KUKA KRL program: MyProgram_152().src

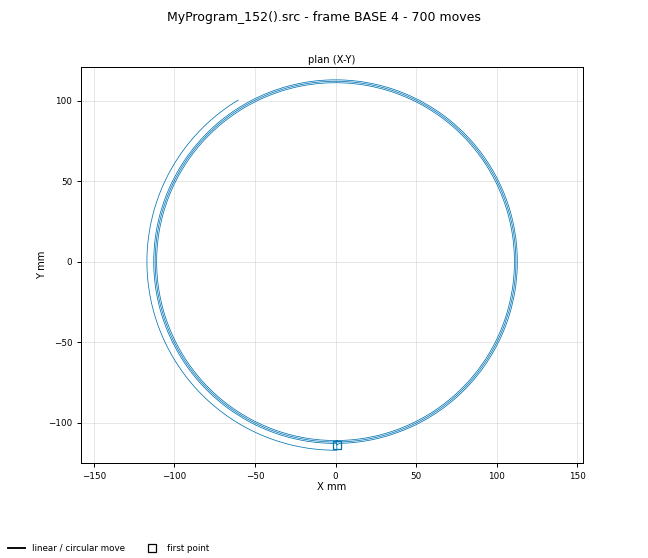
[picture p0: tool path of MyProgram_152().src in frame BASE 4, 700 of 700 moves have a stored position in this frame; points joined in program order, loops and branches not executed]
&ACCESS RVP
&REL 1
&PARAM TEMPLATE = C:\KRC\Roboter\Template\vorgabe
&PARAM EDITMASK = *
DEF MyProgram_152()
; ---- Setting reference (Base) ----
$BASE = BASE_DATA[4]

; --------------------------
; ---- Setting tool (TCP) ----
$TOOL = TOOL_DATA[3]
; --------------------------

$VEL.CP = VEL_APROX_PRINT
LIN {X 0.8048,Y -113.7717,Z 118,A -93.5748,B 24.9556,C -1.539,E1 25.0005,E2 539.5686} C_DIS
Startdeposition()
$VEL.CP = VEL_PRINT
LIN {X 2.402,Y -112.8589,Z 118,A -92.1297,B 24.9531,C -1.5823,E1 25.0048,E2 538.0211} C_DIS
LIN {X 9.2872,Y -112.5017,Z 118,A -88.8373,B 24.9535,C -1.5747,E1 25.014,E2 534.748} C_DIS
LIN {X 15.0576,Y -111.8766,Z 118,A -85.7735,B 24.9531,C -1.5815,E1 25.0225,E2 531.6701} C_DIS
LIN {X 17.7675,Y -111.4782,Z 118,A -84.0166,B 24.9521,C -1.5987,E1 25.0275,E2 529.8742} C_DIS
LIN {X 21.9684,Y -110.727,Z 118,A -81.6298,B 24.9514,C -1.6103,E1 25.0341,E2 527.4627} C_DIS
LIN {X 25.6031,Y -109.9423,Z 118,A -80.4099,B 24.9531,C -1.5825,E1 25.0372,E2 526.3104} C_DIS
LIN {X 28.0521,Y -109.3429,Z 118,A -78.9806,B 24.9526,C -1.5904,E1 25.0411,E2 524.8645} C_DIS
LIN {X 31.4481,Y -108.4172,Z 118,A -77.0293,B 24.9521,C -1.5997,E1 25.0464,E2 522.8944} C_DIS
LIN {X 34.8547,Y -107.3683,Z 118,A -75.3553,B 24.9523,C -1.5959,E1 25.0508,E2 521.2326} C_DIS
LIN {X 42.209,Y -104.6964,Z 118,A -70.4589,B 24.9494,C -1.643,E1 25.0639,E2 516.2353} C_DIS
LIN {X 47.5182,Y -102.3955,Z 118,A -68.4504,B 24.9517,C -1.6055,E1 25.0687,E2 514.3206} C_DIS
LIN {X 50.4487,Y -100.9844,Z 118,A -66.7644,B 24.9514,C -1.6098,E1 25.073,E2 512.6289} C_DIS
LIN {X 54.4638,Y -98.8775,Z 118,A -64.3708,B 24.9509,C -1.6179,E1 25.0789,E2 510.2228} C_DIS
LIN {X 57.7854,Y -96.9732,Z 118,A -62.5355,B 24.951,C -1.6166,E1 25.0833,E2 508.3961} C_DIS
LIN {X 62.6769,Y -93.8871,Z 118,A -59.5043,B 24.9504,C -1.6267,E1 25.0904,E2 505.3512} C_DIS
LIN {X 66.3277,Y -91.3435,Z 118,A -57.343,B 24.9504,C -1.627,E1 25.0953,E2 503.1967} C_DIS
LIN {X 69.139,Y -89.2339,Z 118,A -55.545,B 24.9501,C -1.6315,E1 25.0993,E2 501.3946} C_DIS
LIN {X 72.1712,Y -86.7993,Z 118,A -53.7011,B 24.9502,C -1.63,E1 25.1033,E2 499.5613} C_DIS
LIN {X 75.0077,Y -84.361,Z 118,A -51.7648,B 24.9498,C -1.6361,E1 25.1074,E2 497.6182} C_DIS
LIN {X 77.4909,Y -82.0853,Z 118,A -50.0402,B 24.9495,C -1.6409,E1 25.1109,E2 495.8893} C_DIS
LIN {X 80.3457,Y -79.2929,Z 118,A -48.1006,B 24.9495,C -1.6418,E1 25.1147,E2 493.9557} C_DIS
LIN {X 82.9222,Y -76.5954,Z 118,A -46.1586,B 24.9491,C -1.6488,E1 25.1185,E2 492.0056} C_DIS
LIN {X 85.1759,Y -74.0805,Z 118,A -44.45,B 24.9488,C -1.653,E1 25.1216,E2 490.2948} C_DIS
LIN {X 87.7234,Y -71.045,Z 118,A -42.5175,B 24.9487,C -1.6548,E1 25.125,E2 488.3671} C_DIS
LIN {X 89.93,Y -68.2326,Z 118,A -40.2028,B 24.9469,C -1.6828,E1 25.1291,E2 485.9971} C_DIS
LIN {X 92.1441,Y -65.2094,Z 118,A -38.7629,B 24.9479,C -1.6667,E1 25.1313,E2 484.6022} C_DIS
LIN {X 93.913,Y -62.6378,Z 118,A -36.957,B 24.947,C -1.6814,E1 25.1342,E2 482.7706} C_DIS
LIN {X 97.4321,Y -57.009,Z 118,A -33.6398,B 24.9466,C -1.6888,E1 25.139,E2 479.453} C_DIS
LIN {X 99.7325,Y -52.8802,Z 118,A -31.4879,B 24.9468,C -1.6844,E1 25.1418,E2 477.3226} C_DIS
LIN {X 101.2277,Y -49.9579,Z 118,A -29.5164,B 24.9456,C -1.7037,E1 25.1443,E2 475.3163} C_DIS
LIN {X 102.6063,Y -47.0654,Z 118,A -28.3237,B 24.9466,C -1.6884,E1 25.1457,E2 474.166} C_DIS
LIN {X 104.8738,Y -41.7679,Z 118,A -25.458,B 24.9462,C -1.6947,E1 25.1488,E2 471.3012} C_DIS
LIN {X 106.2374,Y -38.167,Z 118,A -23.2124,B 24.9449,C -1.7143,E1 25.151,E2 469.0218} C_DIS
LIN {X 107.3896,Y -34.7888,Z 118,A -21.1915,B 24.9439,C -1.7299,E1 25.1528,E2 466.9758} C_DIS
LIN {X 108.4193,Y -31.441,Z 118,A -19.8783,B 24.945,C -1.7138,E1 25.1538,E2 465.7079} C_DIS
LIN {X 109.206,Y -28.5851,Z 118,A -18.2604,B 24.9443,C -1.724,E1 25.155,E2 464.0754} C_DIS
LIN {X 110.7265,Y -21.9741,Z 118,A -14.9879,B 24.9441,C -1.7271,E1 25.1569,E2 460.8146} C_DIS
LIN {X 111.2835,Y -18.9442,Z 118,A -12.6628,B 24.9414,C -1.7678,E1 25.1581,E2 458.4071} C_DIS
LIN {X 111.9687,Y -14.3469,Z 118,A -11.195,B 24.9437,C -1.7338,E1 25.1586,E2 457.0282} C_DIS
LIN {X 112.5918,Y -8.1329,Z 118,A -7.7881,B 24.9423,C -1.7551,E1 25.1595,E2 453.5913} C_DIS
LIN {X 112.8314,Y -3.4445,Z 118,A -5.521,B 24.9421,C -1.7575,E1 25.1597,E2 451.332} C_DIS
LIN {X 112.8355,Y 3.3128,Z 118,A -2.3964,B 24.9423,C -1.7544,E1 25.1597,E2 448.2331} C_DIS
LIN {X 112.4849,Y 9.4978,Z 118,A 1.2273,B 24.9402,C -1.7867,E1 25.1591,E2 444.5547} C_DIS
LIN {X 111.9004,Y 14.8741,Z 118,A 3.3995,B 24.9413,C -1.769,E1 25.1584,E2 442.4373} C_DIS
LIN {X 110.8233,Y 21.4709,Z 118,A 6.9455,B 24.9402,C -1.7867,E1 25.1568,E2 438.8703} C_DIS
LIN {X 110.0173,Y 25.2787,Z 118,A 9.1167,B 24.9391,C -1.8019,E1 25.1555,E2 436.6758} C_DIS
LIN {X 109.2742,Y 28.3194,Z 118,A 10.7684,B 24.9386,C -1.8098,E1 25.1543,E2 435.0151} C_DIS
LIN {X 108.2461,Y 32.0247,Z 118,A 12.6004,B 24.9386,C -1.8102,E1 25.1529,E2 433.1925} C_DIS
LIN {X 107.2377,Y 35.2583,Z 118,A 14.4309,B 24.9379,C -1.8206,E1 25.1513,E2 431.348} C_DIS
LIN {X 106.0351,Y 38.7215,Z 118,A 16.7948,B 24.9359,C -1.8495,E1 25.149,E2 428.9292} C_DIS
LIN {X 104.4434,Y 42.8307,Z 118,A 18.3058,B 24.9377,C -1.8225,E1 25.1475,E2 427.4902} C_DIS
LIN {X 103.2018,Y 45.7454,Z 118,A 20.7862,B 24.9346,C -1.8674,E1 25.1446,E2 424.9173} C_DIS
LIN {X 101.0515,Y 50.3133,Z 118,A 22.435,B 24.9371,C -1.8325,E1 25.1427,E2 423.3598} C_DIS
LIN {X 99.7775,Y 52.7948,Z 118,A 23.9415,B 24.9365,C -1.8406,E1 25.1407,E2 421.8421} C_DIS
LIN {X 97.9208,Y 56.1633,Z 118,A 25.9476,B 24.936,C -1.8484,E1 25.138,E2 419.828} C_DIS
LIN {X 95.8852,Y 59.5727,Z 118,A 27.942,B 24.9356,C -1.8528,E1 25.1351,E2 417.8334} C_DIS
LIN {X 92.3072,Y 64.9818,Z 118,A 31.0938,B 24.9356,C -1.8549,E1 25.1302,E2 414.6923} C_DIS
LIN {X 90.1594,Y 67.9272,Z 118,A 33.0026,B 24.935,C -1.8622,E1 25.127,E2 412.7754} C_DIS
LIN {X 86.6208,Y 72.386,Z 118,A 35.9947,B 24.9342,C -1.8738,E1 25.1217,E2 409.7699} C_DIS
LIN {X 84.1132,Y 75.2846,Z 118,A 37.797,B 24.9343,C -1.8718,E1 25.1184,E2 407.9804} C_DIS
LIN {X 80.5166,Y 79.1199,Z 118,A 40.2597,B 24.9346,C -1.8684,E1 25.1138,E2 405.5364} C_DIS
LIN {X 78.3916,Y 81.2253,Z 118,A 42.9434,B 24.9306,C -1.9244,E1 25.1081,E2 402.7315} C_DIS
LIN {X 74.0748,Y 85.1809,Z 118,A 44.7694,B 24.9338,C -1.8785,E1 25.1045,E2 401.0213} C_DIS
LIN {X 72.1339,Y 86.8303,Z 118,A 46.2087,B 24.9332,C -1.8876,E1 25.1014,E2 399.5661} C_DIS
LIN {X 69.1536,Y 89.2227,Z 118,A 48.1804,B 24.9329,C -1.8926,E1 25.0971,E2 397.5899} C_DIS
LIN {X 66.4944,Y 91.2214,Z 118,A 49.8899,B 24.9326,C -1.8965,E1 25.0932,E2 395.8772} C_DIS
LIN {X 64.1479,Y 92.8868,Z 118,A 51.3138,B 24.9326,C -1.8974,E1 25.09,E2 394.4562} C_DIS
LIN {X 59.5117,Y 95.9233,Z 118,A 54.2532,B 24.9318,C -1.9074,E1 25.083,E2 391.5025} C_DIS
LIN {X 53.645,Y 99.323,Z 118,A 57.4079,B 24.9323,C -1.8996,E1 25.0755,E2 388.3757} C_DIS
LIN {X 51.2302,Y 100.5897,Z 118,A 58.9815,B 24.9316,C -1.9098,E1 25.0715,E2 386.7823} C_DIS
LIN {X 46.0651,Y 103.0579,Z 118,A 61.9291,B 24.9312,C -1.9151,E1 25.064,E2 383.8298} C_DIS
LIN {X 42.496,Y 104.5796,Z 118,A 63.7957,B 24.9314,C -1.9127,E1 25.0592,E2 381.9732} C_DIS
LIN {X 39.615,Y 105.7053,Z 118,A 65.4058,B 24.9312,C -1.916,E1 25.055,E2 380.3588} C_DIS
LIN {X 35.9326,Y 107.0124,Z 118,A 67.2162,B 24.9316,C -1.9102,E1 25.0503,E2 378.5657} C_DIS
LIN {X 33.2398,Y 107.8793,Z 118,A 68.6966,B 24.9314,C -1.9133,E1 25.0463,E2 377.0808} C_DIS
LIN {X 29.9302,Y 108.845,Z 118,A 70.5732,B 24.9309,C -1.92,E1 25.0413,E2 375.1914} C_DIS
LIN {X 26.6578,Y 109.6912,Z 118,A 72.2249,B 24.931,C -1.9182,E1 25.0368,E2 373.5462} C_DIS
LIN {X 22.4715,Y 110.625,Z 118,A 74.3991,B 24.931,C -1.9192,E1 25.0309,E2 371.3726} C_DIS
LIN {X 17.7694,Y 111.4779,Z 118,A 76.7319,B 24.9312,C -1.916,E1 25.0245,E2 369.0497} C_DIS
LIN {X 14.5712,Y 111.9396,Z 118,A 78.4355,B 24.9309,C -1.9192,E1 25.0198,E2 367.3401} C_DIS
LIN {X 9.6157,Y 112.4745,Z 118,A 81.4547,B 24.9294,C -1.9405,E1 25.0112,E2 364.2723} C_DIS
LIN {X 5.9662,Y 112.7265,Z 118,A 82.747,B 24.9312,C -1.9163,E1 25.0078,E2 363.0378} C_DIS
LIN {X 2.8641,Y 112.8492,Z 118,A 84.6566,B 24.9301,C -1.9303,E1 25.0024,E2 361.0954} C_DIS
LIN {X -1.9154,Y 112.8679,Z 118,A 87.225,B 24.9297,C -1.9359,E1 24.9952,E2 358.5138} C_DIS
LIN {X -5.2556,Y 112.7623,Z 118,A 88.5128,B 24.931,C -1.918,E1 24.9917,E2 357.2681} C_DIS
LIN {X -8.8083,Y 112.54,Z 118,A 90.828,B 24.9295,C -1.9387,E1 24.9851,E2 354.9028} C_DIS
LIN {X -12.5825,Y 112.1819,Z 118,A 92.1951,B 24.9313,C -1.9142,E1 24.9815,E2 353.5932} C_DIS
LIN {X -17.3713,Y 111.5395,Z 118,A 94.693,B 24.9313,C -1.9145,E1 24.9746,E2 351.0925} C_DIS
LIN {X -20.3299,Y 111.0388,Z 118,A 96.3775,B 24.9309,C -1.9201,E1 24.9699,E2 349.3931} C_DIS
LIN {X -25.507,Y 109.9645,Z 118,A 98.8966,B 24.9315,C -1.9108,E1 24.9631,E2 346.8928} C_DIS
LIN {X -28.5025,Y 109.2272,Z 118,A 100.6115,B 24.9312,C -1.9155,E1 24.9584,E2 345.1644} C_DIS
LIN {X -32.1742,Y 108.2018,Z 118,A 103.4922,B 24.9285,C -1.9529,E1 24.9504,E2 342.1899} C_DIS
LIN {X -38.0694,Y 106.273,Z 118,A 105.533,B 24.9321,C -1.9028,E1 24.9453,E2 340.2643} C_DIS
LIN {X -42.4764,Y 104.5876,Z 118,A 108.4339,B 24.9309,C -1.9204,E1 24.9377,E2 337.3154} C_DIS
LIN {X -45.7728,Y 103.1896,Z 118,A 109.7639,B 24.9325,C -1.8976,E1 24.9344,E2 336.0364} C_DIS
LIN {X -49.0695,Y 101.6613,Z 118,A 111.5813,B 24.9328,C -1.8936,E1 24.9298,E2 334.2237} C_DIS
LIN {X -51.5093,Y 100.447,Z 118,A 113.0723,B 24.9326,C -1.8957,E1 24.9261,E2 332.7237} C_DIS
LIN {X -55.0243,Y 98.5653,Z 118,A 115.45,B 24.9318,C -1.9067,E1 24.9202,E2 330.3131} C_DIS
LIN {X -60.0139,Y 95.6095,Z 118,A 117.963,B 24.9335,C -1.8837,E1 24.9143,E2 327.8472} C_DIS
LIN {X -62.6085,Y 93.9324,Z 118,A 119.8363,B 24.9328,C -1.893,E1 24.9099,E2 325.9456} C_DIS
LIN {X -65.5576,Y 91.8967,Z 118,A 121.5338,B 24.9334,C -1.8844,E1 24.906,E2 324.2627} C_DIS
LIN {X -69.28,Y 89.1252,Z 118,A 123.7333,B 24.9342,C -1.8731,E1 24.9012,E2 322.0822} C_DIS
LIN {X -72.5359,Y 86.4948,Z 118,A 126.1485,B 24.9337,C -1.8801,E1 24.8959,E2 319.6411} C_DIS
LIN {X -76.0629,Y 83.4101,Z 118,A 128.5833,B 24.934,C -1.8769,E1 24.8908,E2 317.2043} C_DIS
LIN {X -79.6121,Y 80.0305,Z 118,A 131.7137,B 24.9325,C -1.8968,E1 24.8845,E2 314.0131} C_DIS
LIN {X -83.2929,Y 76.1913,Z 118,A 133.2341,B 24.9364,C -1.8427,E1 24.8818,E2 312.6152} C_DIS
LIN {X -86.5197,Y 72.5069,Z 118,A 135.9504,B 24.9362,C -1.8453,E1 24.8768,E2 309.8802} C_DIS
LIN {X -87.774,Y 70.9827,Z 118,A 138.0793,B 24.9332,C -1.8879,E1 24.8729,E2 307.6398} C_DIS
LIN {X -91.4324,Y 66.2063,Z 118,A 140.4206,B 24.9358,C -1.8508,E1 24.8692,E2 305.3757} C_DIS
LIN {X -93.4841,Y 63.2733,Z 118,A 142.0112,B 24.9368,C -1.8368,E1 24.8667,E2 303.8107} C_DIS
LIN {X -95.6275,Y 59.9851,Z 118,A 144.3877,B 24.9361,C -1.8464,E1 24.8631,E2 301.3993} C_DIS
LIN {X -97.4074,Y 57.0508,Z 118,A 145.8594,B 24.9372,C -1.8306,E1 24.861,E2 299.9576} C_DIS
LIN {X -100.1802,Y 52.0301,Z 118,A 148.5711,B 24.9383,C -1.8141,E1 24.8575,E2 297.271} C_DIS
LIN {X -102.045,Y 48.271,Z 118,A 151.3144,B 24.9371,C -1.8319,E1 24.8541,E2 294.4701} C_DIS
LIN {X -103.5717,Y 44.8971,Z 118,A 152.6729,B 24.9389,C -1.8056,E1 24.8526,E2 293.167} C_DIS
LIN {X -104.9573,Y 41.5553,Z 118,A 154.5864,B 24.9391,C -1.8029,E1 24.8506,E2 291.2491} C_DIS
LIN {X -106.1713,Y 38.3481,Z 118,A 156.2658,B 24.9396,C -1.7951,E1 24.849,E2 289.5789} C_DIS
LIN {X -107.7159,Y 33.7671,Z 118,A 158.5561,B 24.9406,C -1.781,E1 24.847,E2 287.3093} C_DIS
LIN {X -108.8956,Y 29.7429,Z 118,A 160.9448,B 24.9403,C -1.7844,E1 24.8451,E2 284.8985} C_DIS
LIN {X -109.7388,Y 26.4629,Z 118,A 162.7339,B 24.9405,C -1.7817,E1 24.8439,E2 283.1055} C_DIS
LIN {X -110.5858,Y 22.662,Z 118,A 164.6641,B 24.9411,C -1.7735,E1 24.8428,E2 281.1834} C_DIS
LIN {X -111.2944,Y 18.8792,Z 118,A 166.7269,B 24.9411,C -1.7715,E1 24.8418,E2 279.1132} C_DIS
LIN {X -111.8828,Y 15.0094,Z 118,A 168.8445,B 24.9413,C -1.7702,E1 24.841,E2 276.986} C_DIS
LIN {X -112.4298,Y 10.1196,Z 118,A 171.0591,B 24.9425,C -1.7509,E1 24.8403,E2 274.8041} C_DIS
LIN {X -112.6679,Y 7.0079,Z 118,A 172.789,B 24.9425,C -1.7515,E1 24.84,E2 273.0625} C_DIS
LIN {X -112.8514,Y 2.7946,Z 118,A 175.0901,B 24.9425,C -1.7508,E1 24.8398,E2 270.749} C_DIS
LIN {X -112.8798,Y -1.066,Z 118,A 176.9598,B 24.9432,C -1.741,E1 24.8398,E2 268.8916} C_DIS
LIN {X -112.7664,Y -5.161,Z 118,A 178.8983,B 24.944,C -1.7287,E1 24.84,E2 266.9708} C_DIS
LIN {X -112.5129,Y -9.1472,Z 118,A -178.8825,B 24.944,C -1.7297,E1 24.8405,E2 264.7357} C_DIS
LIN {X -112.1261,Y -13.059,Z 118,A -177.007,B 24.9446,C -1.7186,E1 24.841,E2 262.8755} C_DIS
LIN {X -111.7014,Y -16.3024,Z 118,A -175.2397,B 24.9447,C -1.7175,E1 24.8417,E2 261.1003} C_DIS
LIN {X -111.1154,Y -19.9038,Z 118,A -173.4712,B 24.9453,C -1.7084,E1 24.8425,E2 259.3431} C_DIS
LIN {X -110.5241,Y -22.9629,Z 118,A -171.8012,B 24.9454,C -1.7069,E1 24.8435,E2 257.6667} C_DIS
LIN {X -109.6741,Y -26.7281,Z 118,A -169.9321,B 24.946,C -1.6972,E1 24.8446,E2 255.8097} C_DIS
LIN {X -108.7888,Y -30.1371,Z 118,A -167.9676,B 24.946,C -1.6987,E1 24.8461,E2 253.8302} C_DIS
LIN {X -107.0117,Y -35.9347,Z 118,A -165.0822,B 24.947,C -1.6817,E1 24.8485,E2 250.9687} C_DIS
LIN {X -105.2192,Y -40.8887,Z 118,A -162.5083,B 24.9478,C -1.6698,E1 24.851,E2 248.4088} C_DIS
LIN {X -103.7561,Y -44.4741,Z 118,A -160.2487,B 24.9474,C -1.6757,E1 24.8534,E2 246.1225} C_DIS
LIN {X -102.4324,Y -47.4388,Z 118,A -158.6803,B 24.9479,C -1.6679,E1 24.8552,E2 244.5642} C_DIS
LIN {X -101.025,Y -50.3668,Z 118,A -157.0388,B 24.9482,C -1.6629,E1 24.8572,E2 242.9257} C_DIS
LIN {X -97.8978,Y -56.2034,Z 118,A -153.6518,B 24.9487,C -1.6547,E1 24.8618,E2 239.5404} C_DIS
LIN {X -96.0419,Y -59.3218,Z 118,A -151.1233,B 24.9473,C -1.6775,E1 24.8656,E2 236.9445} C_DIS
LIN {X -93.6226,Y -63.0688,Z 118,A -149.5738,B 24.9494,C -1.6427,E1 24.8678,E2 235.4702} C_DIS
LIN {X -91.8778,Y -65.584,Z 118,A -147.6358,B 24.9487,C -1.6544,E1 24.871,E2 233.495} C_DIS
LIN {X -89.0738,Y -69.3467,Z 118,A -145.5092,B 24.9497,C -1.6381,E1 24.8746,E2 231.3969} C_DIS
LIN {X -86.8469,Y -72.1139,Z 118,A -143.7672,B 24.9501,C -1.6314,E1 24.8776,E2 229.6628} C_DIS
LIN {X -84.7005,Y -74.6248,Z 118,A -141.5087,B 24.9489,C -1.6513,E1 24.8819,E2 227.3467} C_DIS
LIN {X -82.0149,Y -77.5658,Z 118,A -140.1222,B 24.9508,C -1.6208,E1 24.8844,E2 226.0267} C_DIS
LIN {X -80.0918,Y -79.5499,Z 118,A -137.9549,B 24.949,C -1.6492,E1 24.8888,E2 223.7827} C_DIS
LIN {X -76.7997,Y -82.7346,Z 118,A -136.3613,B 24.9512,C -1.6143,E1 24.8919,E2 222.2657} C_DIS
LIN {X -74.3555,Y -84.9357,Z 118,A -134.5873,B 24.9512,C -1.6153,E1 24.8956,E2 220.4823} C_DIS
LIN {X -71.7058,Y -87.186,Z 118,A -132.8472,B 24.9514,C -1.6109,E1 24.8994,E2 218.746} C_DIS
LIN {X -68.9835,Y -89.3537,Z 118,A -131.0718,B 24.9515,C -1.608,E1 24.9033,E2 216.9708} C_DIS
LIN {X -66.1284,Y -91.4894,Z 118,A -128.5939,B 24.9501,C -1.6326,E1 24.909,E2 214.4257} C_DIS
LIN {X -62.517,Y -93.9927,Z 118,A -126.9408,B 24.9517,C -1.6049,E1 24.9127,E2 212.833} C_DIS
LIN {X -56.1542,Y -97.9261,Z 118,A -123.4102,B 24.9527,C -1.5881,E1 24.9211,E2 209.3314} C_DIS
LIN {X -53.8233,Y -99.2263,Z 118,A -121.8335,B 24.9523,C -1.5955,E1 24.925,E2 207.7326} C_DIS
LIN {X -49.1494,Y -101.6229,Z 118,A -119.3373,B 24.9529,C -1.585,E1 24.9311,E2 205.2546} C_DIS
LIN {X -46.4402,Y -102.8888,Z 118,A -117.6708,B 24.9527,C -1.5895,E1 24.9354,E2 203.5734} C_DIS
LIN {X -43.2764,Y -104.2597,Z 118,A -116.0265,B 24.953,C -1.5832,E1 24.9396,E2 201.9402} C_DIS
LIN {X -40.73,Y -105.2811,Z 118,A -114.3179,B 24.9523,C -1.5952,E1 24.9441,E2 200.1996} C_DIS
LIN {X -37.1946,Y -106.5805,Z 118,A -112.6543,B 24.953,C -1.583,E1 24.9484,E2 198.5615} C_DIS
LIN {X -34.6718,Y -107.4275,Z 118,A -111.2175,B 24.9529,C -1.5856,E1 24.9523,E2 197.116} C_DIS
LIN {X -31.0242,Y -108.5374,Z 118,A -109.2871,B 24.9529,C -1.584,E1 24.9574,E2 195.1861} C_DIS
LIN {X -27.9038,Y -109.381,Z 118,A -107.5699,B 24.9529,C -1.5863,E1 24.9621,E2 193.4609} C_DIS
LIN {X -23.577,Y -110.3955,Z 118,A -105.0237,B 24.9522,C -1.5976,E1 24.9691,E2 190.8846} C_DIS
LIN {X -20.4377,Y -111.0194,Z 118,A -103.7543,B 24.9531,C -1.5818,E1 24.9725,E2 189.6514} C_DIS
LIN {X -17.117,Y -111.5788,Z 118,A -101.7896,B 24.9525,C -1.5923,E1 24.978,E2 187.66} C_DIS
LIN {X -13.4063,Y -112.0854,Z 118,A -99.4156,B 24.9513,C -1.6125,E1 24.9847,E2 185.2364} C_DIS
LIN {X -8.5933,Y -112.5572,Z 118,A -98.0495,B 24.9541,C -1.5652,E1 24.9882,E2 183.9819} C_DIS
LIN {X -3.0225,Y -112.8444,Z 118,A -95.0742,B 24.9537,C -1.5715,E1 24.9966,E2 180.9909} C_DIS
LIN {X 0.8049,Y -112.8587,Z 118,A -93.673,B 24.9551,C -1.5489,E1 25.0004,E2 179.6433} C_DIS
Enddeposition()
LIN {X 0.8049,Y -112.8587,Z 118,A -93.673,B 24.9551,C -1.5489,E1 25.0004,E2 179.6433} C_DIS
Startdeposition()
$VEL.CP = VEL_PRINT
LIN {X -0.5745,Y -111.9858,Z 118,A -94.7709,B 24.9551,C -1.5476,E1 24.9972,E2 180.7444} C_DIS
LIN {X -3.7868,Y -111.9237,Z 118,A -96.157,B 24.9545,C -1.5582,E1 24.9934,E2 182.1055} C_DIS
LIN {X -7.5135,Y -111.7348,Z 118,A -97.9421,B 24.9542,C -1.5634,E1 24.9885,E2 183.8788} C_DIS
LIN {X -11.5098,Y -111.3942,Z 118,A -100.191,B 24.9547,C -1.5552,E1 24.9822,E2 186.1482} C_DIS
LIN {X -15.7787,Y -110.87,Z 118,A -102.2228,B 24.9542,C -1.5627,E1 24.9766,E2 188.1637} C_DIS
LIN {X -19.3475,Y -110.3043,Z 118,A -104.1198,B 24.9543,C -1.5613,E1 24.9714,E2 190.066} C_DIS
LIN {X -23.1813,Y -109.5634,Z 118,A -106.2386,B 24.9546,C -1.557,E1 24.9655,E2 192.1973} C_DIS
LIN {X -27.1085,Y -108.6581,Z 118,A -108.2436,B 24.9544,C -1.5605,E1 24.9601,E2 194.1968} C_DIS
LIN {X -30.6703,Y -107.7055,Z 118,A -110.0059,B 24.954,C -1.5669,E1 24.9554,E2 195.9466} C_DIS
LIN {X -33.9607,Y -106.715,Z 118,A -111.8642,B 24.9542,C -1.564,E1 24.9504,E2 197.8149} C_DIS
LIN {X -37.7056,Y -105.4507,Z 118,A -114.3104,B 24.9551,C -1.5484,E1 24.9439,E2 200.3031} C_DIS
LIN {X -41.1518,Y -104.1523,Z 118,A -115.4083,B 24.9531,C -1.5825,E1 24.9412,E2 201.3224} C_DIS
LIN {X -43.7938,Y -103.0696,Z 118,A -117.2802,B 24.954,C -1.5671,E1 24.9363,E2 203.2352} C_DIS
LIN {X -47.1869,Y -101.5605,Z 118,A -119.1288,B 24.9537,C -1.5713,E1 24.9316,E2 205.0782} C_DIS
LIN {X -51.5542,Y -99.4169,Z 118,A -121.7086,B 24.9537,C -1.5707,E1 24.9251,E2 207.6663} C_DIS
LIN {X -55.1785,Y -97.452,Z 118,A -124.0864,B 24.9542,C -1.5628,E1 24.9193,E2 210.0699} C_DIS
LIN {X -57.997,Y -95.7993,Z 118,A -125.3917,B 24.9532,C -1.5801,E1 24.9162,E2 211.338} C_DIS
LIN {X -61.2053,Y -93.7833,Z 118,A -127.3136,B 24.953,C -1.5838,E1 24.9117,E2 213.2573} C_DIS
LIN {X -63.7925,Y -92.0417,Z 118,A -128.989,B 24.953,C -1.5832,E1 24.9078,E2 214.9397} C_DIS
LIN {X -67.2856,Y -89.5197,Z 118,A -131.1116,B 24.9526,C -1.5903,E1 24.9031,E2 217.0529} C_DIS
LIN {X -70.3055,Y -87.1684,Z 118,A -133.0806,B 24.9524,C -1.5935,E1 24.8988,E2 219.0217} C_DIS
LIN {X -72.836,Y -85.0654,Z 118,A -134.8178,B 24.9524,C -1.5946,E1 24.895,E2 220.763} C_DIS
LIN {X -75.5524,Y -82.662,Z 118,A -136.5759,B 24.9519,C -1.6022,E1 24.8914,E2 222.51} C_DIS
LIN {X -78.3741,Y -79.9927,Z 118,A -138.6634,B 24.9519,C -1.6023,E1 24.8872,E2 224.6058} C_DIS
LIN {X -80.7054,Y -77.6387,Z 118,A -140.3339,B 24.9516,C -1.607,E1 24.8839,E2 226.2724} C_DIS
LIN {X -83.5821,Y -74.5332,Z 118,A -142.5561,B 24.9515,C -1.6096,E1 24.8797,E2 228.4982} C_DIS
LIN {X -86.1435,Y -71.5572,Z 118,A -144.5627,B 24.9512,C -1.6144,E1 24.8761,E2 230.5025} C_DIS
LIN {X -88.6006,Y -68.4916,Z 118,A -146.5521,B 24.9508,C -1.6201,E1 24.8727,E2 232.4878} C_DIS
LIN {X -90.2439,Y -66.3114,Z 118,A -148.0471,B 24.9508,C -1.6196,E1 24.8702,E2 233.991} C_DIS
LIN {X -92.6156,Y -62.9565,Z 118,A -150.1693,B 24.9506,C -1.6242,E1 24.8668,E2 236.1128} C_DIS
LIN {X -94.7497,Y -59.6976,Z 118,A -152.1219,B 24.9502,C -1.631,E1 24.8639,E2 238.0591} C_DIS
LIN {X -96.5814,Y -56.6857,Z 118,A -153.8752,B 24.9497,C -1.6378,E1 24.8614,E2 239.8052} C_DIS
LIN {X -98.0921,Y -54.0322,Z 118,A -155.7655,B 24.9503,C -1.6292,E1 24.8588,E2 241.7259} C_DIS
LIN {X -100.272,Y -49.8665,Z 118,A -157.9152,B 24.9492,C -1.6459,E1 24.8561,E2 243.8473} C_DIS
LIN {X -101.9518,Y -46.3367,Z 118,A -159.9324,B 24.9489,C -1.6509,E1 24.8537,E2 245.8636} C_DIS
LIN {X -103.325,Y -43.1876,Z 118,A -161.6252,B 24.9485,C -1.6586,E1 24.8518,E2 247.5475} C_DIS
LIN {X -104.5495,Y -40.1347,Z 118,A -163.5115,B 24.9486,C -1.6556,E1 24.8499,E2 249.4514} C_DIS
LIN {X -105.999,Y -36.1312,Z 118,A -165.56,B 24.9479,C -1.6672,E1 24.848,E2 251.484} C_DIS
LIN {X -106.8545,Y -33.5167,Z 118,A -167.1419,B 24.9481,C -1.6647,E1 24.8467,E2 253.0809} C_DIS
LIN {X -108.0405,Y -29.4694,Z 118,A -169.1564,B 24.9473,C -1.6768,E1 24.8451,E2 255.0781} C_DIS
LIN {X -108.8878,Y -26.1674,Z 118,A -170.8539,B 24.9469,C -1.684,E1 24.844,E2 256.7683} C_DIS
LIN {X -109.6214,Y -22.9005,Z 118,A -172.6695,B 24.9468,C -1.6855,E1 24.8429,E2 258.5913} C_DIS
LIN {X -110.3093,Y -19.3198,Z 118,A -174.55,B 24.9464,C -1.6908,E1 24.842,E2 260.4703} C_DIS
LIN {X -110.8494,Y -15.9234,Z 118,A -176.2651,B 24.946,C -1.6981,E1 24.8413,E2 262.1781} C_DIS
LIN {X -111.2706,Y -12.6536,Z 118,A -177.9242,B 24.9456,C -1.7045,E1 24.8407,E2 263.8318} C_DIS
LIN {X -111.598,Y -9.3378,Z 118,A -179.7404,B 24.9455,C -1.7057,E1 24.8402,E2 265.656} C_DIS
LIN {X -111.8556,Y -5.4657,Z 118,A 178.2813,B 24.945,C -1.7124,E1 24.8399,E2 267.6304} C_DIS
LIN {X -111.9651,Y -2.231,Z 118,A 176.6126,B 24.9447,C -1.7173,E1 24.8398,E2 269.2974} C_DIS
LIN {X -111.9776,Y 1.5512,Z 118,A 174.8422,B 24.9439,C -1.7299,E1 24.8398,E2 271.0484} C_DIS
LIN {X -111.881,Y 4.876,Z 118,A 172.9941,B 24.9439,C -1.7299,E1 24.84,E2 272.9079} C_DIS
LIN {X -111.6848,Y 8.2517,Z 118,A 171.1815,B 24.9438,C -1.7322,E1 24.8403,E2 274.7255} C_DIS
LIN {X -111.3826,Y 11.6206,Z 118,A 169.5019,B 24.9433,C -1.7398,E1 24.8408,E2 276.3971} C_DIS
LIN {X -110.9169,Y 15.4488,Z 118,A 167.5976,B 24.9427,C -1.7489,E1 24.8414,E2 278.2913} C_DIS
LIN {X -110.4747,Y 18.3433,Z 118,A 165.9806,B 24.9427,C -1.7492,E1 24.8422,E2 279.9171} C_DIS
LIN {X -109.8458,Y 21.8044,Z 118,A 164.1468,B 24.9424,C -1.7537,E1 24.8431,E2 281.7511} C_DIS
LIN {X -109.1224,Y 25.1679,Z 118,A 162.3485,B 24.9421,C -1.7579,E1 24.8442,E2 283.5499} C_DIS
LIN {X -108.1283,Y 29.1446,Z 118,A 160.3258,B 24.9415,C -1.7674,E1 24.8456,E2 285.5616} C_DIS
LIN {X -107.1457,Y 32.5777,Z 118,A 158.3203,B 24.9415,C -1.7664,E1 24.8472,E2 287.5812} C_DIS
LIN {X -105.8884,Y 36.4573,Z 118,A 156.2404,B 24.9411,C -1.7732,E1 24.8491,E2 289.6568} C_DIS
LIN {X -104.4949,Y 40.2788,Z 118,A 154.1306,B 24.9407,C -1.7785,E1 24.8511,E2 291.7657} C_DIS
LIN {X -102.9647,Y 44.0427,Z 118,A 152.0569,B 24.9403,C -1.7851,E1 24.8534,E2 293.8351} C_DIS
LIN {X -101.0823,Y 48.2038,Z 118,A 149.8146,B 24.9396,C -1.7959,E1 24.856,E2 296.0641} C_DIS
LIN {X -99.5426,Y 51.3084,Z 118,A 147.6251,B 24.9403,C -1.7852,E1 24.8588,E2 298.2909} C_DIS
LIN {X -97.9282,Y 54.3257,Z 118,A 146.3056,B 24.9388,C -1.8069,E1 24.8605,E2 299.5656} C_DIS
LIN {X -96.6613,Y 56.5506,Z 118,A 144.7331,B 24.9392,C -1.8006,E1 24.8627,E2 301.1613} C_DIS
LIN {X -94.4253,Y 60.2088,Z 118,A 142.7578,B 24.9382,C -1.8153,E1 24.8656,E2 303.1116} C_DIS
LIN {X -92.6598,Y 62.8912,Z 118,A 141.129,B 24.9379,C -1.8204,E1 24.8681,E2 304.7363} C_DIS
LIN {X -90.9222,Y 65.3793,Z 118,A 139.2074,B 24.9386,C -1.8105,E1 24.8713,E2 306.6909} C_DIS
LIN {X -87.9402,Y 69.3373,Z 118,A 136.97,B 24.9373,C -1.8288,E1 24.8751,E2 308.8952} C_DIS
LIN {X -85.9631,Y 71.7742,Z 118,A 134.9228,B 24.9382,C -1.816,E1 24.8788,E2 310.9825} C_DIS
LIN {X -83.6204,Y 74.4904,Z 118,A 133.4962,B 24.9368,C -1.8365,E1 24.8814,E2 312.3667} C_DIS
LIN {X -79.125,Y 79.251,Z 118,A 130.2685,B 24.9359,C -1.8495,E1 24.8876,E2 315.5773} C_DIS
LIN {X -74.6518,Y 83.476,Z 118,A 127.1896,B 24.9352,C -1.8597,E1 24.8938,E2 318.6447} C_DIS
LIN {X -71.6538,Y 86.0632,Z 118,A 124.9775,B 24.9354,C -1.8569,E1 24.8985,E2 320.8719} C_DIS
LIN {X -68.9681,Y 88.232,Z 118,A 122.7135,B 24.9365,C -1.8412,E1 24.9036,E2 323.1815} C_DIS
LIN {X -66.1165,Y 90.3866,Z 118,A 121.3273,B 24.935,C -1.8624,E1 24.9066,E2 324.5223} C_DIS
LIN {X -63.0509,Y 92.5517,Z 118,A 119.403,B 24.9347,C -1.8661,E1 24.911,E2 326.4444} C_DIS
LIN {X -60.2796,Y 94.3799,Z 118,A 117.8526,B 24.9341,C -1.8753,E1 24.9146,E2 327.978} C_DIS
LIN {X -55.5698,Y 97.2275,Z 118,A 114.7971,B 24.9344,C -1.8709,E1 24.922,E2 331.0532} C_DIS
LIN {X -52.3376,Y 99.0047,Z 118,A 112.9869,B 24.9339,C -1.8772,E1 24.9264,E2 332.8535} C_DIS
LIN {X -49.1692,Y 100.6177,Z 118,A 110.9539,B 24.9343,C -1.8716,E1 24.9315,E2 334.9052} C_DIS
LIN {X -46.014,Y 102.0972,Z 118,A 108.7584,B 24.9353,C -1.858,E1 24.9372,E2 337.1384} C_DIS
LIN {X -42.045,Y 103.7949,Z 118,A 107.1533,B 24.9334,C -1.8851,E1 24.9412,E2 338.6826} C_DIS
LIN {X -38.5911,Y 105.128,Z 118,A 105.2252,B 24.9334,C -1.8863,E1 24.9462,E2 340.612} C_DIS
LIN {X -35.8646,Y 106.0889,Z 118,A 103.4354,B 24.9341,C -1.8756,E1 24.9511,E2 342.4305} C_DIS
LIN {X -30.803,Y 107.6679,Z 118,A 101.0128,B 24.933,C -1.8903,E1 24.9574,E2 344.8223} C_DIS
LIN {X -27.1503,Y 108.648,Z 118,A 99.2166,B 24.9325,C -1.8979,E1 24.9623,E2 346.6032} C_DIS
LIN {X -24.015,Y 109.382,Z 118,A 97.4918,B 24.9325,C -1.8962,E1 24.967,E2 348.3341} C_DIS
LIN {X -20.5011,Y 110.0968,Z 118,A 95.4668,B 24.933,C -1.89,E1 24.9726,E2 350.3762} C_DIS
LIN {X -16.8382,Y 110.7144,Z 118,A 93.6372,B 24.9327,C -1.8942,E1 24.9776,E2 352.1974} C_DIS
LIN {X -13.2487,Y 111.2009,Z 118,A 91.7678,B 24.9327,C -1.8947,E1 24.9828,E2 354.067} C_DIS
LIN {X -9.0521,Y 111.6208,Z 118,A 89.6543,B 24.9325,C -1.8976,E1 24.9886,E2 356.1747} C_DIS
LIN {X -4.9987,Y 111.8757,Z 118,A 87.6218,B 24.9323,C -1.9002,E1 24.9943,E2 358.2015} C_DIS
LIN {X -0.6033,Y 111.9856,Z 118,A 85.3405,B 24.9323,C -1.8995,E1 25.0007,E2 360.4847} C_DIS
LIN {X 3.222,Y 111.941,Z 118,A 83.5015,B 24.932,C -1.9046,E1 25.0058,E2 362.3112} C_DIS
LIN {X 6.04,Y 111.8243,Z 118,A 81.8881,B 24.9325,C -1.8976,E1 25.0103,E2 363.9408} C_DIS
LIN {X 10.352,Y 111.5077,Z 118,A 79.7606,B 24.9323,C -1.901,E1 25.0162,E2 366.0592} C_DIS
LIN {X 14.0678,Y 111.1005,Z 118,A 77.9049,B 24.9321,C -1.903,E1 25.0213,E2 367.9087} C_DIS
LIN {X 16.9124,Y 110.7029,Z 118,A 76.4246,B 24.9321,C -1.9021,E1 25.0254,E2 369.3897} C_DIS
LIN {X 20.3817,Y 110.1183,Z 118,A 74.5073,B 24.9326,C -1.8965,E1 25.0307,E2 371.3183} C_DIS
LIN {X 23.9362,Y 109.3992,Z 118,A 72.7644,B 24.9323,C -1.9004,E1 25.0355,E2 373.0497} C_DIS
LIN {X 27.4732,Y 108.5658,Z 118,A 70.8534,B 24.9325,C -1.8971,E1 25.0407,E2 374.9658} C_DIS
LIN {X 31.1674,Y 107.5647,Z 118,A 68.8013,B 24.9329,C -1.8918,E1 25.0462,E2 377.027} C_DIS
LIN {X 35.058,Y 106.3599,Z 118,A 66.3131,B 24.9342,C -1.873,E1 25.0529,E2 379.555} C_DIS
LIN {X 38.7212,Y 105.0806,Z 118,A 64.8821,B 24.9327,C -1.8947,E1 25.0565,E2 380.9318} C_DIS
LIN {X 42.1989,Y 103.7322,Z 118,A 62.9916,B 24.9327,C -1.8935,E1 25.0614,E2 382.8208} C_DIS
LIN {X 45.0529,Y 102.5254,Z 118,A 61.4223,B 24.9329,C -1.8925,E1 25.0655,E2 384.3889} C_DIS
LIN {X 48.538,Y 100.9217,Z 118,A 59.4242,B 24.9331,C -1.8886,E1 25.0705,E2 386.391} C_DIS
LIN {X 51.9415,Y 99.2133,Z 118,A 57.7336,B 24.9325,C -1.8972,E1 25.0747,E2 388.0567} C_DIS
LIN {X 56.9022,Y 96.4535,Z 118,A 54.621,B 24.9335,C -1.884,E1 25.0823,E2 391.1911} C_DIS
LIN {X 59.6373,Y 94.7874,Z 118,A 52.7085,B 24.9345,C -1.8696,E1 25.0869,E2 393.1317} C_DIS
LIN {X 63.3045,Y 92.38,Z 118,A 50.6656,B 24.9341,C -1.8746,E1 25.0916,E2 395.1558} C_DIS
LIN {X 65.9718,Y 90.4925,Z 118,A 49.0406,B 24.9341,C -1.8738,E1 25.0953,E2 396.7772} C_DIS
LIN {X 68.3876,Y 88.6807,Z 118,A 47.4945,B 24.9344,C -1.871,E1 25.0987,E2 398.3243} C_DIS
LIN {X 71.2379,Y 86.4088,Z 118,A 45.6242,B 24.9346,C -1.8672,E1 25.1028,E2 400.1965} C_DIS
LIN {X 73.8301,Y 84.2038,Z 118,A 43.2081,B 24.9369,C -1.8344,E1 25.108,E2 402.6806} C_DIS
LIN {X 77.3372,Y 80.9961,Z 118,A 41.428,B 24.9353,C -1.8577,E1 25.1115,E2 404.3983} C_DIS
LIN {X 81.1979,Y 77.1254,Z 118,A 38.6622,B 24.9356,C -1.853,E1 25.1169,E2 407.1634} C_DIS
LIN {X 83.5693,Y 74.5475,Z 118,A 36.8808,B 24.9359,C -1.8494,E1 25.1202,E2 408.9454} C_DIS
LIN {X 86.0348,Y 71.688,Z 118,A 35.1044,B 24.9357,C -1.8517,E1 25.1234,E2 410.7082} C_DIS
LIN {X 88.2868,Y 68.8988,Z 118,A 33.0749,B 24.9366,C -1.8386,E1 25.127,E2 412.7592} C_DIS
LIN {X 90.4188,Y 66.0725,Z 118,A 31.4032,B 24.9366,C -1.8403,E1 25.1297,E2 414.4187} C_DIS
LIN {X 94.7725,Y 59.6612,Z 118,A 27.5639,B 24.9368,C -1.8356,E1 25.1357,E2 418.2502} C_DIS
LIN {X 96.5553,Y 56.7299,Z 118,A 25.5783,B 24.9379,C -1.8206,E1 25.1386,E2 420.2609} C_DIS
LIN {X 98.4833,Y 53.3121,Z 118,A 23.6973,B 24.9379,C -1.8208,E1 25.1411,E2 422.1317} C_DIS
LIN {X 100.1401,Y 50.1326,Z 118,A 21.5918,B 24.939,C -1.8035,E1 25.1438,E2 424.2669} C_DIS
LIN {X 102.077,Y 46.0589,Z 118,A 19.5678,B 24.9386,C -1.8096,E1 25.1462,E2 426.2654} C_DIS
LIN {X 103.4728,Y 42.8363,Z 118,A 17.7259,B 24.9391,C -1.8023,E1 25.1482,E2 428.1146} C_DIS
LIN {X 105.0886,Y 38.6992,Z 118,A 15.4813,B 24.9395,C -1.7969,E1 25.1504,E2 430.3594} C_DIS
LIN {X 106.2602,Y 35.3568,Z 118,A 13.6503,B 24.9399,C -1.7905,E1 25.1521,E2 432.1951} C_DIS
LIN {X 107.353,Y 31.8821,Z 118,A 11.8418,B 24.9401,C -1.7874,E1 25.1536,E2 434.0008} C_DIS
LIN {X 108.3493,Y 28.3153,Z 118,A 9.9588,B 24.9405,C -1.782,E1 25.1549,E2 435.8855} C_DIS
LIN {X 109.1957,Y 24.8508,Z 118,A 8.2044,B 24.9406,C -1.7795,E1 25.1561,E2 437.6357} C_DIS
LIN {X 109.9521,Y 21.2526,Z 118,A 5.9188,B 24.9423,C -1.7554,E1 25.1573,E2 439.9649} C_DIS
LIN {X 110.565,Y 17.803,Z 118,A 4.4097,B 24.9418,C -1.7624,E1 25.158,E2 441.4485} C_DIS
LIN {X 111.0489,Y 14.4661,Z 118,A 2.4377,B 24.9429,C -1.7458,E1 25.1587,E2 443.4481} C_DIS
LIN {X 111.4357,Y 11.1089,Z 118,A 0.9834,B 24.9424,C -1.7526,E1 25.1591,E2 444.8776} C_DIS
LIN {X 111.8002,Y 6.4759,Z 118,A -1.2499,B 24.9425,C -1.7515,E1 25.1596,E2 447.1003} C_DIS
LIN {X 111.9418,Y 3.1958,Z 118,A -3.3028,B 24.944,C -1.7291,E1 25.1598,E2 449.1938} C_DIS
LIN {X 111.9875,Y -0.1098,Z 118,A -4.7829,B 24.9437,C -1.7332,E1 25.1598,E2 450.6555} C_DIS
LIN {X 111.9008,Y -4.4159,Z 118,A -6.7721,B 24.9435,C -1.7357,E1 25.1596,E2 452.6269} C_DIS
LIN {X 111.7335,Y -7.5333,Z 118,A -8.3663,B 24.9439,C -1.7307,E1 25.1593,E2 454.2235} C_DIS
LIN {X 111.3241,Y -12.1798,Z 118,A -10.8752,B 24.9447,C -1.7173,E1 25.1587,E2 456.749} C_DIS
LIN {X 110.7098,Y -16.868,Z 118,A -13.0682,B 24.9446,C -1.7197,E1 25.1578,E2 458.9234} C_DIS
LIN {X 110.2658,Y -19.5614,Z 118,A -14.5327,B 24.9451,C -1.7121,E1 25.1571,E2 460.3973} C_DIS
LIN {X 109.5725,Y -23.1384,Z 118,A -16.6722,B 24.9463,C -1.6936,E1 25.1559,E2 462.5681} C_DIS
LIN {X 108.513,Y -27.6784,Z 118,A -18.7658,B 24.9459,C -1.6992,E1 25.1546,E2 464.6363} C_DIS
LIN {X 107.5806,Y -31.1114,Z 118,A -20.9028,B 24.9472,C -1.6789,E1 25.1529,E2 466.8088} C_DIS
LIN {X 105.2063,Y -38.3765,Z 118,A -24.552,B 24.9472,C -1.6785,E1 25.1497,E2 470.4385} C_DIS
LIN {X 103.9074,Y -41.7682,Z 118,A -26.4438,B 24.9477,C -1.6712,E1 25.1477,E2 472.3371} C_DIS
LIN {X 102.2148,Y -45.753,Z 118,A -28.5116,B 24.9477,C -1.671,E1 25.1454,E2 474.3938} C_DIS
LIN {X 100.5788,Y -49.2476,Z 118,A -30.4742,B 24.948,C -1.6656,E1 25.1431,E2 476.3589} C_DIS
LIN {X 99.1203,Y -52.1182,Z 118,A -32.0902,B 24.9482,C -1.6621,E1 25.141,E2 477.9745} C_DIS
LIN {X 97.5594,Y -54.9862,Z 118,A -33.6882,B 24.9483,C -1.6604,E1 25.1388,E2 479.568} C_DIS
LIN {X 93.9782,Y -60.9054,Z 118,A -37.3857,B 24.9494,C -1.643,E1 25.1334,E2 483.2878} C_DIS
LIN {X 89.6426,Y -67.122,Z 118,A -41.1385,B 24.9497,C -1.6378,E1 25.1273,E2 487.0345} C_DIS
LIN {X 87.4183,Y -69.9971,Z 118,A -43.0879,B 24.9503,C -1.6288,E1 25.1239,E2 488.9962} C_DIS
LIN {X 85.1381,Y -72.7506,Z 118,A -44.8622,B 24.9504,C -1.6264,E1 25.1208,E2 490.7679} C_DIS
LIN {X 82.6524,Y -75.5628,Z 118,A -46.719,B 24.9506,C -1.6243,E1 25.1173,E2 492.6213} C_DIS
LIN {X 80.1717,Y -78.1925,Z 118,A -48.6312,B 24.951,C -1.6169,E1 25.1136,E2 494.5429} C_DIS
LIN {X 77.7678,Y -80.5811,Z 118,A -50.255,B 24.951,C -1.6176,E1 25.1104,E2 496.1582} C_DIS
LIN {X 75.2674,Y -82.9235,Z 118,A -52.1252,B 24.9515,C -1.6082,E1 25.1065,E2 498.0431} C_DIS
LIN {X 72.7166,Y -85.1671,Z 118,A -53.7395,B 24.9515,C -1.6097,E1 25.1031,E2 499.6474} C_DIS
LIN {X 69.9272,Y -87.474,Z 118,A -55.698,B 24.952,C -1.6008,E1 25.0988,E2 501.6195} C_DIS
LIN {X 67.047,Y -89.699,Z 118,A -57.3427,B 24.9516,C -1.6065,E1 25.0952,E2 503.2448} C_DIS
LIN {X 63.1255,Y -92.5012,Z 118,A -60.6962,B 24.9543,C -1.5623,E1 25.0873,E2 506.6913} C_DIS
LIN {X 58.8007,Y -95.31,Z 118,A -62.5916,B 24.9526,C -1.5898,E1 25.083,E2 508.5156} C_DIS
LIN {X 54.8704,Y -97.6241,Z 118,A -64.883,B 24.9528,C -1.5874,E1 25.0775,E2 510.8057} C_DIS
LIN {X 51.5583,Y -99.4149,Z 118,A -66.9098,B 24.9532,C -1.5796,E1 25.0724,E2 512.8451} C_DIS
LIN {X 47.8408,Y -101.2561,Z 118,A -68.7955,B 24.9528,C -1.5866,E1 25.0677,E2 514.7094} C_DIS
LIN {X 44.1406,Y -102.9232,Z 118,A -71.0642,B 24.9535,C -1.575,E1 25.0619,E2 517} C_DIS
LIN {X 40.8297,Y -104.2788,Z 118,A -72.829,B 24.9535,C -1.5753,E1 25.0573,E2 518.7602} C_DIS
LIN {X 35.8555,Y -106.092,Z 118,A -75.483,B 24.9535,C -1.5741,E1 25.0504,E2 521.4115} C_DIS
LIN {X 32.3764,Y -107.2063,Z 118,A -77.3824,B 24.9538,C -1.5706,E1 25.0453,E2 523.3158} C_DIS
LIN {X 29.1659,Y -108.1225,Z 118,A -79.0337,B 24.9538,C -1.5712,E1 25.0408,E2 524.963} C_DIS
LIN {X 25.647,Y -109.0117,Z 118,A -81.0371,B 24.9542,C -1.563,E1 25.0354,E2 526.9829} C_DIS
LIN {X 21.022,Y -109.9965,Z 118,A -83.3407,B 24.9541,C -1.5659,E1 25.0291,E2 529.2769} C_DIS
LIN {X 17.3728,Y -110.6317,Z 118,A -85.2301,B 24.9541,C -1.5646,E1 25.0239,E2 531.1671} C_DIS
LIN {X 14.3317,Y -111.0663,Z 118,A -87.0597,B 24.9548,C -1.5526,E1 25.0188,E2 533.0238} C_DIS
LIN {X 9.4082,Y -111.5923,Z 118,A -89.5103,B 24.9548,C -1.5547,E1 25.012,E2 535.4678} C_DIS
LIN {X 4.8498,Y -111.8821,Z 118,A -91.6426,B 24.9543,C -1.5625,E1 25.0061,E2 537.581} C_DIS
LIN {X 1.8855,Y -111.9714,Z 118,A -93.346,B 24.9547,C -1.5541,E1 25.0013,E2 539.3039} C_DIS
LIN {X 1.8855,Y -111.9714,Z 118,A -93.346,B 24.9547,C -1.5541,E1 25.0013,E2 539.3039} C_DIS
Enddeposition()
LIN {X 0.7947,Y -111.0873,Z 118,A -93.4382,B 24.9527,C -1.5895,E1 25.0013,E2 539.3122} C_DIS
Startdeposition()
$VEL.CP = VEL_PRINT
LIN {X 4.083,Y -111.0173,Z 118,A -91.3466,B 24.9516,C -1.6068,E1 25.0072,E2 537.18} C_DIS
LIN {X 6.7943,Y -110.8844,Z 118,A -89.9479,B 24.9516,C -1.6073,E1 25.0111,E2 535.7805} C_DIS
LIN {X 9.5001,Y -110.6853,Z 118,A -88.5496,B 24.9516,C -1.608,E1 25.015,E2 534.3815} C_DIS
LIN {X 12.2305,Y -110.417,Z 118,A -87.1367,B 24.9516,C -1.6087,E1 25.0189,E2 532.9678} C_DIS
LIN {X 14.9524,Y -110.0816,Z 118,A -85.7248,B 24.9515,C -1.6095,E1 25.0228,E2 531.5552} C_DIS
LIN {X 17.6388,Y -109.6831,Z 118,A -84.3257,B 24.9515,C -1.6105,E1 25.0267,E2 530.1552} C_DIS
LIN {X 20.314,Y -109.2192,Z 118,A -82.9277,B 24.9513,C -1.6115,E1 25.0305,E2 528.7562} C_DIS
LIN {X 22.9755,Y -108.6904,Z 118,A -81.5307,B 24.9513,C -1.6126,E1 25.0343,E2 527.3583} C_DIS
LIN {X 25.4287,Y -108.1417,Z 118,A -80.2194,B 24.9512,C -1.6145,E1 25.0379,E2 526.0443} C_DIS
LIN {X 28.3085,Y -107.4251,Z 118,A -78.7097,B 24.9512,C -1.6152,E1 25.042,E2 524.5354} C_DIS
LIN {X 30.931,Y -106.6995,Z 118,A -77.3097,B 24.951,C -1.6166,E1 25.0458,E2 523.1343} C_DIS
LIN {X 33.5346,Y -105.91,Z 118,A -75.91,B 24.951,C -1.6181,E1 25.0495,E2 521.7336} C_DIS
LIN {X 36.0817,Y -105.0693,Z 118,A -74.1982,B 24.95,C -1.6343,E1 25.0541,E2 519.9869} C_DIS
LIN {X 39.9906,Y -103.6449,Z 118,A -72.3944,B 24.9507,C -1.6221,E1 25.0588,E2 518.2156} C_DIS
LIN {X 42.5078,Y -102.6382,Z 118,A -70.9969,B 24.9506,C -1.6241,E1 25.0624,E2 516.8166} C_DIS
LIN {X 44.9992,Y -101.5705,Z 118,A -69.6036,B 24.9505,C -1.626,E1 25.0659,E2 515.4222} C_DIS
LIN {X 47.4977,Y -100.4266,Z 118,A -68.191,B 24.9503,C -1.6281,E1 25.0695,E2 514.0084} C_DIS
LIN {X 49.9415,Y -99.2339,Z 118,A -66.7933,B 24.9503,C -1.6302,E1 25.073,E2 512.6095} C_DIS
LIN {X 52.355,Y -97.9819,Z 118,A -65.3963,B 24.9501,C -1.6324,E1 25.0765,E2 511.2112} C_DIS
LIN {X 54.7365,Y -96.6717,Z 118,A -63.9999,B 24.9499,C -1.6346,E1 25.0799,E2 509.8135} C_DIS
LIN {X 57.1188,Y -95.2836,Z 118,A -62.5865,B 24.9498,C -1.6369,E1 25.0833,E2 508.3992} C_DIS
LIN {X 59.4073,Y -93.8736,Z 118,A -61.203,B 24.9496,C -1.6394,E1 25.0866,E2 507.0141} C_DIS
LIN {X 61.6544,Y -92.413,Z 118,A -59.8273,B 24.9495,C -1.6419,E1 25.0898,E2 505.6372} C_DIS
LIN {X 64.3775,Y -90.5353,Z 118,A -57.9736,B 24.9489,C -1.652,E1 25.094,E2 503.7659} C_DIS
LIN {X 67.6949,Y -88.0823,Z 118,A -55.9714,B 24.9489,C -1.6509,E1 25.0985,E2 501.7735} C_DIS
LIN {X 70.2038,Y -86.0965,Z 118,A -54.2014,B 24.9484,C -1.66,E1 25.1024,E2 499.9889} C_DIS
LIN {X 73.0752,Y -83.6725,Z 118,A -52.439,B 24.9486,C -1.6565,E1 25.1061,E2 498.2414} C_DIS
LIN {X 75.1035,Y -81.8568,Z 118,A -50.9865,B 24.9482,C -1.662,E1 25.1091,E2 496.7818} C_DIS
LIN {X 77.8282,Y -79.2714,Z 118,A -49.0188,B 24.9479,C -1.6681,E1 25.1131,E2 494.808} C_DIS
LIN {X 79.9861,Y -77.0928,Z 118,A -47.4802,B 24.9477,C -1.6701,E1 25.1161,E2 493.2713} C_DIS
LIN {X 82.0911,Y -74.8481,Z 118,A -45.8125,B 24.9473,C -1.6777,E1 25.1192,E2 491.5928} C_DIS
LIN {X 84.5559,Y -72.0511,Z 118,A -44.0488,B 24.9473,C -1.6756,E1 25.1224,E2 489.8422} C_DIS
LIN {X 86.5115,Y -69.6918,Z 118,A -42.4755,B 24.9471,C -1.6795,E1 25.1252,E2 488.267} C_DIS
LIN {X 88.2115,Y -67.5272,Z 118,A -41.0383,B 24.9469,C -1.6841,E1 25.1277,E2 486.8256} C_DIS
LIN {X 90.0591,Y -65.0449,Z 118,A -39.4871,B 24.9467,C -1.6865,E1 25.1302,E2 485.2763} C_DIS
LIN {X 91.6139,Y -62.8363,Z 118,A -38.1015,B 24.9465,C -1.69,E1 25.1325,E2 483.8891} C_DIS
LIN {X 93.1157,Y -60.5887,Z 118,A -36.7104,B 24.9462,C -1.6938,E1 25.1346,E2 482.496} C_DIS
LIN {X 94.5616,Y -58.3061,Z 118,A -35.3256,B 24.946,C -1.6975,E1 25.1366,E2 481.1097} C_DIS
LIN {X 95.9486,Y -55.9939,Z 118,A -33.943,B 24.9458,C -1.7012,E1 25.1386,E2 479.7254} C_DIS
LIN {X 97.3272,Y -53.5624,Z 118,A -32.5124,B 24.9455,C -1.7049,E1 25.1406,E2 478.2934} C_DIS
LIN {X 98.7741,Y -50.8414,Z 118,A -30.8511,B 24.945,C -1.713,E1 25.1427,E2 476.6219} C_DIS
LIN {X 100.1141,Y -48.1481,Z 118,A -29.3869,B 24.945,C -1.7137,E1 25.1445,E2 475.1638} C_DIS
LIN {X 101.2686,Y -45.6699,Z 118,A -27.9908,B 24.9447,C -1.7173,E1 25.1461,E2 473.7666} C_DIS
LIN {X 102.3779,Y -43.1258,Z 118,A -26.5833,B 24.9445,C -1.7207,E1 25.1477,E2 472.3591} C_DIS
LIN {X 103.4149,Y -40.5763,Z 118,A -25.1043,B 24.9441,C -1.7278,E1 25.1492,E2 470.8715} C_DIS
LIN {X 104.579,Y -37.479,Z 118,A -23.4625,B 24.9439,C -1.7301,E1 25.1508,E2 469.2333} C_DIS
LIN {X 105.442,Y -34.9764,Z 118,A -21.9507,B 24.9432,C -1.7411,E1 25.1522,E2 467.704} C_DIS
LIN {X 106.5171,Y -31.5462,Z 118,A -20.2037,B 24.9432,C -1.7422,E1 25.1536,E2 465.9646} C_DIS
LIN {X 107.4231,Y -28.3162,Z 118,A -18.5458,B 24.943,C -1.7444,E1 25.1548,E2 464.3111} C_DIS
LIN {X 108.0844,Y -25.6766,Z 118,A -17.1518,B 24.9427,C -1.7484,E1 25.1557,E2 462.9155} C_DIS
LIN {X 108.6858,Y -22.9982,Z 118,A -15.7482,B 24.9424,C -1.7525,E1 25.1565,E2 461.5106} C_DIS
LIN {X 109.2157,Y -20.3338,Z 118,A -14.3549,B 24.9422,C -1.7566,E1 25.1573,E2 460.1155} C_DIS
LIN {X 109.6801,Y -17.6573,Z 118,A -12.9633,B 24.9419,C -1.7608,E1 25.1579,E2 458.7225} C_DIS
LIN {X 110.1199,Y -14.6566,Z 118,A -11.3087,B 24.9413,C -1.77,E1 25.1586,E2 457.0558} C_DIS
LIN {X 110.4886,Y -11.5468,Z 118,A -9.7604,B 24.9411,C -1.7722,E1 25.159,E2 455.5115} C_DIS
LIN {X 110.7916,Y -8.1693,Z 118,A -8.0706,B 24.9409,C -1.7752,E1 25.1594,E2 453.8247} C_DIS
LIN {X 110.9581,Y -5.4604,Z 118,A -6.6794,B 24.9407,C -1.7794,E1 25.1596,E2 452.4319} C_DIS
LIN {X 111.0583,Y -2.7489,Z 118,A -5.2895,B 24.9404,C -1.7835,E1 25.1598,E2 451.0405} C_DIS
LIN {X 111.0906,Y -0.1969,Z 118,A -3.9947,B 24.9402,C -1.7868,E1 25.1598,E2 449.7456} C_DIS
LIN {X 111.0631,Y 2.503,Z 118,A -2.5851,B 24.9398,C -1.7921,E1 25.1598,E2 448.3318} C_DIS
LIN {X 110.9591,Y 5.4391,Z 118,A -1.0945,B 24.9395,C -1.7959,E1 25.1595,E2 446.8412} C_DIS
LIN {X 110.7936,Y 8.1399,Z 118,A 0.2911,B 24.9393,C -1.7999,E1 25.1593,E2 445.4543} C_DIS
LIN {X 110.5629,Y 10.8309,Z 118,A 1.6742,B 24.939,C -1.804,E1 25.1589,E2 444.0699} C_DIS
LIN {X 110.2681,Y 13.504,Z 118,A 3.055,B 24.9387,C -1.8081,E1 25.1585,E2 442.6874} C_DIS
LIN {X 109.843,Y 16.6049,Z 118,A 4.7499,B 24.9381,C -1.817,E1 25.1578,E2 440.9816} C_DIS
LIN {X 109.3356,Y 19.6671,Z 118,A 6.2433,B 24.9381,C -1.8172,E1 25.1571,E2 439.4966} C_DIS
LIN {X 108.8153,Y 22.3672,Z 118,A 7.6387,B 24.9379,C -1.8206,E1 25.1563,E2 438.1012} C_DIS
LIN {X 108.2319,Y 25.0386,Z 118,A 9.0403,B 24.9376,C -1.8246,E1 25.1555,E2 436.6983} C_DIS
LIN {X 107.5861,Y 27.6819,Z 118,A 10.4341,B 24.9373,C -1.8285,E1 25.1545,E2 435.3032} C_DIS
LIN {X 106.8759,Y 30.3085,Z 118,A 11.8729,B 24.9369,C -1.8345,E1 25.1534,E2 433.8588} C_DIS
LIN {X 106.0049,Y 33.2286,Z 118,A 13.437,B 24.9366,C -1.8389,E1 25.1522,E2 432.2931} C_DIS
LIN {X 105.0498,Y 36.1395,Z 118,A 14.9747,B 24.9364,C -1.8417,E1 25.1508,E2 430.7574} C_DIS
LIN {X 104.1422,Y 38.6769,Z 118,A 16.3632,B 24.9361,C -1.8458,E1 25.1495,E2 429.3671} C_DIS
LIN {X 103.1463,Y 41.2596,Z 118,A 17.7716,B 24.9359,C -1.8492,E1 25.148,E2 427.9585} C_DIS
LIN {X 102.107,Y 43.7686,Z 118,A 19.1662,B 24.9356,C -1.853,E1 25.1465,E2 426.5626} C_DIS
LIN {X 101.0066,Y 46.2513,Z 118,A 20.558,B 24.9354,C -1.8566,E1 25.1449,E2 425.1698} C_DIS
LIN {X 99.8462,Y 48.7056,Z 118,A 22.0921,B 24.9347,C -1.8666,E1 25.143,E2 423.6203} C_DIS
LIN {X 98.306,Y 51.7396,Z 118,A 23.7077,B 24.9347,C -1.8653,E1 25.141,E2 422.0165} C_DIS
LIN {X 96.9795,Y 54.1853,Z 118,A 25.1057,B 24.9347,C -1.8676,E1 25.1391,E2 420.6204} C_DIS
LIN {X 95.6544,Y 56.4917,Z 118,A 26.4839,B 24.9343,C -1.8716,E1 25.1371,E2 419.2398} C_DIS
LIN {X 94.1505,Y 58.9641,Z 118,A 28.0399,B 24.9339,C -1.8784,E1 25.1349,E2 417.6757} C_DIS
LIN {X 92.4057,Y 61.6654,Z 118,A 29.6173,B 24.9339,C -1.879,E1 25.1324,E2 416.1046} C_DIS
LIN {X 90.9093,Y 63.8503,Z 118,A 31.1308,B 24.9331,C -1.8891,E1 25.13,E2 414.5746} C_DIS
LIN {X 88.8394,Y 66.6981,Z 118,A 32.7896,B 24.9333,C -1.8867,E1 25.1273,E2 412.9296} C_DIS
LIN {X 87.1588,Y 68.8797,Z 118,A 34.259,B 24.9329,C -1.8923,E1 25.1247,E2 411.4538} C_DIS
LIN {X 84.7709,Y 71.7987,Z 118,A 36.2199,B 24.9325,C -1.8976,E1 25.1212,E2 409.4894} C_DIS
LIN {X 82.7712,Y 74.0945,Z 118,A 37.7542,B 24.9324,C -1.8996,E1 25.1184,E2 407.9572} C_DIS
LIN {X 80.2212,Y 76.8488,Z 118,A 39.7113,B 24.932,C -1.9049,E1 25.1146,E2 405.9963} C_DIS
LIN {X 78.0694,Y 79.0331,Z 118,A 41.2539,B 24.9319,C -1.9066,E1 25.1116,E2 404.4562} C_DIS
LIN {X 75.3656,Y 81.6162,Z 118,A 43.2052,B 24.9315,C -1.9116,E1 25.1076,E2 402.5011} C_DIS
LIN {X 73.074,Y 83.6735,Z 118,A 44.7563,B 24.9314,C -1.9131,E1 25.1044,E2 400.9525} C_DIS
LIN {X 70.2043,Y 86.0961,Z 118,A 46.7153,B 24.931,C -1.9178,E1 25.1002,E2 398.9899} C_DIS
LIN {X 67.5372,Y 88.2038,Z 118,A 48.5064,B 24.9307,C -1.9227,E1 25.0962,E2 397.1938} C_DIS
LIN {X 64.5498,Y 90.4123,Z 118,A 50.2811,B 24.9309,C -1.9199,E1 25.0922,E2 395.4321} C_DIS
LIN {X 62.2593,Y 92.0046,Z 118,A 51.7131,B 24.9307,C -1.922,E1 25.0889,E2 394} C_DIS
LIN {X 60.0215,Y 93.4799,Z 118,A 53.1031,B 24.9306,C -1.9245,E1 25.0857,E2 392.6086} C_DIS
LIN {X 57.6742,Y 94.9461,Z 118,A 54.5118,B 24.9305,C -1.9259,E1 25.0823,E2 391.201} C_DIS
LIN {X 55.3445,Y 96.3226,Z 118,A 55.8876,B 24.9304,C -1.9271,E1 25.079,E2 389.8266} C_DIS
LIN {X 53.0392,Y 97.611,Z 118,A 57.2747,B 24.9302,C -1.9301,E1 25.0756,E2 388.4365} C_DIS
LIN {X 50.4238,Y 98.9875,Z 118,A 58.8532,B 24.9298,C -1.9344,E1 25.0717,E2 386.8521} C_DIS
LIN {X 47.5054,Y 100.4229,Z 118,A 60.4553,B 24.9299,C -1.9332,E1 25.0677,E2 385.257} C_DIS
LIN {X 45.0156,Y 101.5634,Z 118,A 61.8636,B 24.9299,C -1.9346,E1 25.0641,E2 383.8488} C_DIS
LIN {X 42.5165,Y 102.6347,Z 118,A 63.2646,B 24.9297,C -1.9361,E1 25.0605,E2 382.4477} C_DIS
LIN {X 39.992,Y 103.6444,Z 118,A 64.6638,B 24.9297,C -1.9374,E1 25.0568,E2 381.0486} C_DIS
LIN {X 37.4359,Y 104.5948,Z 118,A 66.067,B 24.9295,C -1.9385,E1 25.0532,E2 379.6455} C_DIS
LIN {X 34.8857,Y 105.4726,Z 118,A 67.456,B 24.9295,C -1.9396,E1 25.0495,E2 378.2566} C_DIS
LIN {X 31.8105,Y 106.4388,Z 118,A 69.1696,B 24.9292,C -1.9431,E1 25.0449,E2 376.5379} C_DIS
LIN {X 28.9412,Y 107.2542,Z 118,A 70.637,B 24.9294,C -1.9411,E1 25.041,E2 375.0775} C_DIS
LIN {X 26.3055,Y 107.9309,Z 118,A 72.0386,B 24.9294,C -1.9419,E1 25.0372,E2 373.6762} C_DIS
LIN {X 23.6522,Y 108.5433,Z 118,A 73.5162,B 24.929,C -1.9457,E1 25.0331,E2 372.1915} C_DIS
LIN {X 20.3387,Y 109.2147,Z 118,A 75.1988,B 24.9292,C -1.9439,E1 25.0285,E2 370.5154} C_DIS
LIN {X 17.6438,Y 109.6824,Z 118,A 76.6065,B 24.9292,C -1.9442,E1 25.0246,E2 369.1083} C_DIS
LIN {X 14.9555,Y 110.0811,Z 118,A 78.0085,B 24.9292,C -1.9446,E1 25.0208,E2 367.7066} C_DIS
LIN {X 12.2584,Y 110.414,Z 118,A 79.4105,B 24.9291,C -1.9449,E1 25.0169,E2 366.305} C_DIS
LIN {X 9.5548,Y 110.6806,Z 118,A 80.8112,B 24.9291,C -1.9449,E1 25.013,E2 364.9048} C_DIS
LIN {X 6.2923,Y 110.9121,Z 118,A 82.5461,B 24.9289,C -1.9471,E1 25.0081,E2 363.1657} C_DIS
LIN {X 3.3846,Y 111.0388,Z 118,A 83.9837,B 24.9291,C -1.9443,E1 25.0041,E2 361.7351} C_DIS
LIN {X 0.7303,Y 111.088,Z 118,A 85.3825,B 24.9291,C -1.9453,E1 25.0002,E2 360.334} C_DIS
LIN {X -2.0449,Y 111.0715,Z 118,A 86.7844,B 24.9291,C -1.9438,E1 24.9963,E2 358.9358} C_DIS
LIN {X -4.6941,Y 110.9912,Z 118,A 88.1947,B 24.9291,C -1.9451,E1 24.9924,E2 357.522} C_DIS
LIN {X -7.4562,Y 110.8398,Z 118,A 89.5961,B 24.9291,C -1.9435,E1 24.9885,E2 356.1239} C_DIS
LIN {X -10.2266,Y 110.6186,Z 118,A 91.0162,B 24.9293,C -1.9423,E1 24.9845,E2 354.706} C_DIS
LIN {X -12.929,Y 110.3354,Z 118,A 92.439,B 24.9293,C -1.9423,E1 24.9806,E2 353.2822} C_DIS
LIN {X -15.6449,Y 109.9832,Z 118,A 93.8385,B 24.9293,C -1.941,E1 24.9767,E2 351.8849} C_DIS
LIN {X -18.2894,Y 109.5745,Z 118,A 95.2454,B 24.9293,C -1.941,E1 24.9728,E2 350.4764} C_DIS
LIN {X -21.026,Y 109.0824,Z 118,A 96.6675,B 24.9295,C -1.9395,E1 24.9689,E2 349.0566} C_DIS
LIN {X -24.0786,Y 108.4502,Z 118,A 98.2985,B 24.9295,C -1.939,E1 24.9645,E2 347.4248} C_DIS
LIN {X -27.2853,Y 107.6881,Z 118,A 100.0844,B 24.9294,C -1.9409,E1 24.9596,E2 345.632} C_DIS
LIN {X -30.3108,Y 106.8752,Z 118,A 101.5871,B 24.9298,C -1.9346,E1 24.9556,E2 344.1418} C_DIS
LIN {X -32.8609,Y 106.1189,Z 118,A 102.985,B 24.9298,C -1.9341,E1 24.9519,E2 342.7428} C_DIS
LIN {X -35.5345,Y 105.2538,Z 118,A 104.4291,B 24.93,C -1.9321,E1 24.9481,E2 341.3006} C_DIS
LIN {X -38.0008,Y 104.3888,Z 118,A 105.8047,B 24.93,C -1.9315,E1 24.9444,E2 339.9237} C_DIS
LIN {X -40.5729,Y 103.4162,Z 118,A 107.2177,B 24.9302,C -1.9294,E1 24.9408,E2 338.5128} C_DIS
LIN {X -43.0837,Y 102.3956,Z 118,A 108.6199,B 24.9303,C -1.9276,E1 24.9371,E2 337.1118} C_DIS
LIN {X -45.6206,Y 101.2908,Z 118,A 110.0489,B 24.9305,C -1.9255,E1 24.9335,E2 335.6842} C_DIS
LIN {X -48.2274,Y 100.076,Z 118,A 111.6026,B 24.9305,C -1.926,E1 24.9296,E2 334.1253} C_DIS
LIN {X -51.1597,Y 98.6114,Z 118,A 113.2239,B 24.9309,C -1.9204,E1 24.9256,E2 332.513} C_DIS
LIN {X -53.2818,Y 97.4794,Z 118,A 114.4954,B 24.9309,C -1.9196,E1 24.9224,E2 331.24} C_DIS
LIN {X -55.8595,Y 96.0267,Z 118,A 116.1547,B 24.9307,C -1.9221,E1 24.9184,E2 329.5696} C_DIS
LIN {X -58.8314,Y 94.2334,Z 118,A 117.8117,B 24.9314,C -1.9135,E1 24.9145,E2 327.928} C_DIS
LIN {X -61.1188,Y 92.7661,Z 118,A 119.2046,B 24.9316,C -1.9105,E1 24.9112,E2 326.5378} C_DIS
LIN {X -63.4193,Y 91.2088,Z 118,A 120.6438,B 24.9318,C -1.9078,E1 24.9079,E2 325.1} C_DIS
LIN {X -65.63,Y 89.6313,Z 118,A 122.0353,B 24.932,C -1.9046,E1 24.9048,E2 323.7113} C_DIS
LIN {X -67.8139,Y 87.9906,Z 118,A 123.527,B 24.932,C -1.9049,E1 24.9014,E2 322.2136} C_DIS
LIN {X -70.7151,Y 85.6772,Z 118,A 125.4911,B 24.9321,C -1.9026,E1 24.8972,E2 320.2474} C_DIS
LIN {X -73.314,Y 83.4639,Z 118,A 127.2991,B 24.9323,C -1.9005,E1 24.8934,E2 318.4374} C_DIS
LIN {X -76.0524,Y 80.9759,Z 118,A 129.1642,B 24.9327,C -1.8943,E1 24.8896,E2 316.5794} C_DIS
LIN {X -78.7761,Y 78.3296,Z 118,A 131.1462,B 24.933,C -1.8905,E1 24.8856,E2 314.5983} C_DIS
LIN {X -81.1196,Y 75.8996,Z 118,A 132.9494,B 24.9331,C -1.8886,E1 24.8822,E2 312.7917} C_DIS
LIN {X -83.6128,Y 73.1435,Z 118,A 134.8113,B 24.9336,C -1.8816,E1 24.8787,E2 310.9383} C_DIS
LIN {X -86.0998,Y 70.1996,Z 118,A 136.8138,B 24.934,C -1.8769,E1 24.8751,E2 308.9376} C_DIS
LIN {X -88.203,Y 67.5383,Z 118,A 138.5137,B 24.9344,C -1.8703,E1 24.8722,E2 307.2454} C_DIS
LIN {X -90.0145,Y 65.1066,Z 118,A 140.0548,B 24.9348,C -1.8651,E1 24.8697,E2 305.7093} C_DIS
LIN {X -91.6091,Y 62.8434,Z 118,A 141.4918,B 24.935,C -1.8615,E1 24.8674,E2 304.2738} C_DIS
LIN {X -93.1201,Y 60.5819,Z 118,A 142.9045,B 24.9353,C -1.8579,E1 24.8652,E2 302.8625} C_DIS
LIN {X -94.5753,Y 58.2841,Z 118,A 144.3162,B 24.9356,C -1.8542,E1 24.8632,E2 301.4524} C_DIS
LIN {X -95.9827,Y 55.9361,Z 118,A 145.7352,B 24.9358,C -1.8504,E1 24.8611,E2 300.0351} C_DIS
LIN {X -97.3175,Y 53.5801,Z 118,A 147.2646,B 24.9358,C -1.8515,E1 24.8591,E2 298.4952} C_DIS
LIN {X -98.8872,Y 50.62,Z 118,A 148.9244,B 24.9363,C -1.8437,E1 24.8569,E2 296.845} C_DIS
LIN {X -100.4019,Y 47.5492,Z 118,A 150.6699,B 24.9367,C -1.8376,E1 24.8548,E2 295.1047} C_DIS
LIN {X -101.5682,Y 45.0045,Z 118,A 152.1106,B 24.937,C -1.8331,E1 24.8532,E2 293.6668} C_DIS
LIN {X -102.6391,Y 42.5058,Z 118,A 153.5223,B 24.9373,C -1.8292,E1 24.8516,E2 292.2567} C_DIS
LIN {X -103.5729,Y 40.1738,Z 118,A 154.8407,B 24.9375,C -1.826,E1 24.8503,E2 290.9382} C_DIS
LIN {X -104.5959,Y 37.4329,Z 118,A 156.3476,B 24.9378,C -1.8212,E1 24.8488,E2 289.4344} C_DIS
LIN {X -105.4805,Y 34.8623,Z 118,A 157.7591,B 24.9381,C -1.8172,E1 24.8476,E2 288.0244} C_DIS
LIN {X -106.3016,Y 32.2717,Z 118,A 159.1705,B 24.9384,C -1.8132,E1 24.8464,E2 286.6145} C_DIS
LIN {X -107.1412,Y 29.3597,Z 118,A 160.8566,B 24.9384,C -1.8129,E1 24.8451,E2 284.9191} C_DIS
LIN {X -107.9341,Y 26.2924,Z 118,A 162.3747,B 24.9391,C -1.8033,E1 24.8441,E2 283.4153} C_DIS
LIN {X -108.5458,Y 23.6406,Z 118,A 163.7882,B 24.9393,C -1.7991,E1 24.8433,E2 282.0033} C_DIS
LIN {X -109.0808,Y 21.0343,Z 118,A 165.1844,B 24.9396,C -1.7956,E1 24.8425,E2 280.6073} C_DIS
LIN {X -109.6009,Y 18.1316,Z 118,A 166.7563,B 24.9398,C -1.7927,E1 24.8418,E2 279.033} C_DIS
LIN {X -110.0821,Y 14.9486,Z 118,A 168.3926,B 24.9402,C -1.7863,E1 24.8411,E2 277.4021} C_DIS
LIN {X -110.4164,Y 12.2369,Z 118,A 169.8067,B 24.9405,C -1.782,E1 24.8407,E2 275.99} C_DIS
LIN {X -110.683,Y 9.5289,Z 118,A 171.2199,B 24.9408,C -1.7778,E1 24.8403,E2 274.5783} C_DIS
LIN {X -110.8788,Y 6.8799,Z 118,A 172.602,B 24.941,C -1.7738,E1 24.84,E2 273.1973} C_DIS
LIN {X -111.0168,Y 4.0973,Z 118,A 174.048,B 24.9413,C -1.7695,E1 24.8399,E2 271.753} C_DIS
LIN {X -111.084,Y 1.3671,Z 118,A 175.4928,B 24.9415,C -1.7663,E1 24.8398,E2 270.3071} C_DIS
LIN {X -111.084,Y -1.3665,Z 118,A 176.8847,B 24.9419,C -1.761,E1 24.8398,E2 268.9194} C_DIS
LIN {X -111.0173,Y -4.0858,Z 118,A 178.2992,B 24.9421,C -1.7569,E1 24.8399,E2 267.5061} C_DIS
LIN {X -110.8839,Y -6.8025,Z 118,A 179.7116,B 24.9424,C -1.7528,E1 24.8402,E2 266.0951} C_DIS
LIN {X -110.6841,Y -9.5147,Z 118,A -178.8726,B 24.9427,C -1.7488,E1 24.8405,E2 264.6804} C_DIS
LIN {X -110.4151,Y -12.2483,Z 118,A -177.4509,B 24.943,C -1.7444,E1 24.8409,E2 263.2605} C_DIS
LIN {X -110.0821,Y -14.9483,Z 118,A -176.0364,B 24.9432,C -1.7404,E1 24.8414,E2 261.8472} C_DIS
LIN {X -109.7007,Y -17.5249,Z 118,A -174.6791,B 24.9435,C -1.7367,E1 24.842,E2 260.4906} C_DIS
LIN {X -109.1148,Y -20.8578,Z 118,A -172.8801,B 24.9437,C -1.7333,E1 24.8429,E2 258.6891} C_DIS
LIN {X -108.5446,Y -23.6459,Z 118,A -171.4349,B 24.9441,C -1.7278,E1 24.8437,E2 257.2485} C_DIS
LIN {X -107.9329,Y -26.2975,Z 118,A -170.0218,B 24.9443,C -1.7238,E1 24.8446,E2 255.8365} C_DIS
LIN {X -107.2564,Y -28.9331,Z 118,A -168.5874,B 24.9445,C -1.7207,E1 24.8456,E2 254.4013} C_DIS
LIN {X -106.3029,Y -32.2676,Z 118,A -166.8252,B 24.9449,C -1.7141,E1 24.847,E2 252.6444} C_DIS
LIN {X -105.4832,Y -34.8543,Z 118,A -165.2646,B 24.9449,C -1.7162,E1 24.8484,E2 251.07} C_DIS
LIN {X -104.3783,Y -38.0295,Z 118,A -163.6553,B 24.9454,C -1.7062,E1 24.8499,E2 249.4754} C_DIS
LIN {X -103.4095,Y -40.5899,Z 118,A -162.2336,B 24.9457,C -1.7024,E1 24.8513,E2 248.0548} C_DIS
LIN {X -102.3845,Y -43.1102,Z 118,A -160.8213,B 24.9459,C -1.6987,E1 24.8528,E2 246.6436} C_DIS
LIN {X -101.273,Y -45.6602,Z 118,A -159.4167,B 24.9463,C -1.6934,E1 24.8544,E2 245.2438} C_DIS
LIN {X -100.0553,Y -48.2705,Z 118,A -157.8319,B 24.9463,C -1.693,E1 24.8563,E2 243.6513} C_DIS
LIN {X -98.6113,Y -51.16,Z 118,A -156.2206,B 24.9467,C -1.6862,E1 24.8583,E2 242.0476} C_DIS
LIN {X -97.3176,Y -53.5798,Z 118,A -154.7994,B 24.9469,C -1.6825,E1 24.8602,E2 240.6276} C_DIS
LIN {X -95.9789,Y -55.9426,Z 118,A -153.2373,B 24.9468,C -1.6851,E1 24.8624,E2 239.0513} C_DIS
LIN {X -94.2393,Y -58.822,Z 118,A -151.6297,B 24.9474,C -1.6755,E1 24.8648,E2 237.4583} C_DIS
LIN {X -92.7737,Y -61.1074,Z 118,A -150.2364,B 24.9476,C -1.6716,E1 24.8669,E2 236.0673} C_DIS
LIN {X -91.2651,Y -63.3384,Z 118,A -148.8094,B 24.9478,C -1.6695,E1 24.8691,E2 234.6381} C_DIS
LIN {X -89.6066,Y -65.6637,Z 118,A -147.3718,B 24.9481,C -1.6645,E1 24.8715,E2 233.2057} C_DIS
LIN {X -87.9915,Y -67.8127,Z 118,A -145.9635,B 24.9482,C -1.6619,E1 24.8739,E2 231.7966} C_DIS
LIN {X -86.0988,Y -70.2009,Z 118,A -144.3798,B 24.9484,C -1.6586,E1 24.8766,E2 230.2134} C_DIS
LIN {X -83.909,Y -72.8043,Z 118,A -142.5185,B 24.9484,C -1.6588,E1 24.88,E2 228.3432} C_DIS
LIN {X -81.8481,Y -75.1129,Z 118,A -140.9552,B 24.9487,C -1.6539,E1 24.883,E2 226.7847} C_DIS
LIN {X -79.7392,Y -77.3489,Z 118,A -139.2719,B 24.9487,C -1.6543,E1 24.8862,E2 225.093} C_DIS
LIN {X -77.1022,Y -79.977,Z 118,A -137.4283,B 24.9492,C -1.6472,E1 24.8899,E2 223.2586} C_DIS
LIN {X -74.3396,Y -82.5518,Z 118,A -135.4466,B 24.9493,C -1.6446,E1 24.894,E2 221.2751} C_DIS
LIN {X -71.8004,Y -84.7695,Z 118,A -133.6258,B 24.9493,C -1.6446,E1 24.8978,E2 219.4473} C_DIS
LIN {X -68.8917,Y -87.1493,Z 118,A -131.7859,B 24.9498,C -1.637,E1 24.9018,E2 217.6186} C_DIS
LIN {X -66.1755,Y -89.2318,Z 118,A -130.0741,B 24.9501,C -1.6317,E1 24.9056,E2 215.9133} C_DIS
LIN {X -63.9534,Y -90.8376,Z 118,A -128.6567,B 24.9503,C -1.6294,E1 24.9088,E2 214.4964} C_DIS
LIN {X -61.492,Y -92.5201,Z 118,A -127.0003,B 24.9501,C -1.6317,E1 24.9127,E2 212.8289} C_DIS
LIN {X -58.84,Y -94.228,Z 118,A -125.4432,B 24.9504,C -1.6264,E1 24.9164,E2 211.2796} C_DIS
LIN {X -55.9642,Y -95.9662,Z 118,A -123.7395,B 24.9507,C -1.6226,E1 24.9204,E2 209.5797} C_DIS
LIN {X -53.1654,Y -97.5426,Z 118,A -122.0116,B 24.9507,C -1.6233,E1 24.9247,E2 207.8453} C_DIS
LIN {X -50.5889,Y -98.9031,Z 118,A -120.5672,B 24.9509,C -1.6189,E1 24.9282,E2 206.4072} C_DIS
LIN {X -48.1359,Y -100.1199,Z 118,A -119.1557,B 24.9509,C -1.6172,E1 24.9318,E2 204.9961} C_DIS
LIN {X -45.6707,Y -101.2682,Z 118,A -117.7496,B 24.9511,C -1.6157,E1 24.9354,E2 203.5901} C_DIS
LIN {X -43.1219,Y -102.3795,Z 118,A -116.3268,B 24.9512,C -1.6137,E1 24.939,E2 202.1687} C_DIS
LIN {X -40.5942,Y -103.4078,Z 118,A -114.853,B 24.9512,C -1.6151,E1 24.9428,E2 200.6884} C_DIS
LIN {X -37.4626,Y -104.585,Z 118,A -112.9863,B 24.9509,C -1.6193,E1 24.9478,E2 198.8078} C_DIS
LIN {X -34.1646,Y -105.7064,Z 118,A -111.3726,B 24.9514,C -1.6103,E1 24.952,E2 197.2126} C_DIS
LIN {X -31.5644,Y -106.5118,Z 118,A -109.9809,B 24.9515,C -1.6088,E1 24.9557,E2 195.8221} C_DIS
LIN {X -28.9461,Y -107.2529,Z 118,A -108.5399,B 24.9515,C -1.6095,E1 24.9596,E2 194.3772} C_DIS
LIN {X -25.6766,Y -108.0844,Z 118,A -106.8181,B 24.9515,C -1.6077,E1 24.9643,E2 192.6573} C_DIS
LIN {X -23.0139,Y -108.6825,Z 118,A -105.4093,B 24.9516,C -1.6071,E1 24.9681,E2 191.2482} C_DIS
LIN {X -20.3307,Y -109.2162,Z 118,A -103.999,B 24.9516,C -1.6065,E1 24.972,E2 189.8376} C_DIS
LIN {X -17.6545,Y -109.6806,Z 118,A -102.5955,B 24.9516,C -1.6062,E1 24.9759,E2 188.4336} C_DIS
LIN {X -14.9682,Y -110.0793,Z 118,A -101.1942,B 24.9516,C -1.6059,E1 24.9797,E2 187.0319} C_DIS
LIN {X -12.2742,Y -110.4121,Z 118,A -99.7936,B 24.9516,C -1.6058,E1 24.9836,E2 185.6307} C_DIS
LIN {X -9.5754,Y -110.6787,Z 118,A -98.3941,B 24.9516,C -1.6057,E1 24.9875,E2 184.2307} C_DIS
LIN {X -6.8204,Y -110.8828,Z 118,A -96.97,B 24.9516,C -1.6057,E1 24.9915,E2 182.806} C_DIS
LIN {X -4.1121,Y -111.0162,Z 118,A -95.5717,B 24.9516,C -1.6058,E1 24.9954,E2 181.4072} C_DIS
LIN {X -1.4037,Y -111.0833,Z 118,A -94.1751,B 24.9516,C -1.606,E1 24.9993,E2 180.01} C_DIS
LIN {X 0.7947,Y -111.0873,Z 118,A -93.438,B 24.9527,C -1.5895,E1 25.0012,E2 179.3122} C_DIS
Enddeposition()
LIN {X 0.8233,Y -117.1042,Z 119,A -93.0702,B 24.9574,C -1.5078,E1 25.0017,E2 179.1379} C_DIS
Startdeposition()
$VEL.CP = VEL_PRINT
LIN {X -2.874,Y -117.0753,Z 119,A -95.2834,B 24.9585,C -1.4892,E1 24.9954,E2 181.3951} C_DIS
LIN {X -5.4524,Y -116.9821,Z 119,A -96.5677,B 24.9585,C -1.4882,E1 24.9918,E2 182.6823} C_DIS
LIN {X -8.3217,Y -116.8131,Z 119,A -97.974,B 24.9585,C -1.4882,E1 24.9879,E2 184.0891} C_DIS
LIN {X -11.4788,Y -116.5467,Z 119,A -99.5021,B 24.9585,C -1.4892,E1 24.9837,E2 185.6155} C_DIS
LIN {X -14.0434,Y -116.2641,Z 119,A -100.7871,B 24.9585,C -1.4884,E1 24.9801,E2 186.9032} C_DIS
LIN {X -17.1837,Y -115.843,Z 119,A -102.3156,B 24.9585,C -1.4897,E1 24.9759,E2 188.4299} C_DIS
LIN {X -20.0214,Y -115.3864,Z 119,A -103.7228,B 24.9585,C -1.4901,E1 24.972,E2 189.8376} C_DIS
LIN {X -22.7777,Y -114.8737,Z 119,A -105.0898,B 24.9584,C -1.4908,E1 24.9682,E2 191.2043} C_DIS
LIN {X -25.6591,Y -114.265,Z 119,A -106.538,B 24.9584,C -1.4911,E1 24.9643,E2 192.6535} C_DIS
LIN {X -28.1697,Y -113.6707,Z 119,A -107.8017,B 24.9584,C -1.4918,E1 24.9609,E2 193.9174} C_DIS
LIN {X -31.2349,Y -112.8684,Z 119,A -109.3541,B 24.9583,C -1.4926,E1 24.9567,E2 195.4701} C_DIS
LIN {X -33.9954,Y -112.0678,Z 119,A -110.7625,B 24.9583,C -1.4935,E1 24.9529,E2 196.8787} C_DIS
LIN {X -36.4555,Y -111.2904,Z 119,A -112.0267,B 24.9582,C -1.4944,E1 24.9495,E2 198.1431} C_DIS
LIN {X -39.4534,Y -110.2648,Z 119,A -113.5797,B 24.9581,C -1.4956,E1 24.9454,E2 199.6962} C_DIS
LIN {X -41.8724,Y -109.3675,Z 119,A -114.8293,B 24.958,C -1.4974,E1 24.9422,E2 200.9444} C_DIS
LIN {X -44.8163,Y -108.1961,Z 119,A -116.3981,B 24.958,C -1.4981,E1 24.9381,E2 202.5149} C_DIS
LIN {X -47.1884,Y -107.1812,Z 119,A -117.6803,B 24.958,C -1.4986,E1 24.9348,E2 203.7988} C_DIS
LIN {X -49.6781,Y -106.0497,Z 119,A -119.0495,B 24.958,C -1.4988,E1 24.9313,E2 205.1709} C_DIS
LIN {X -52.6542,Y -104.606,Z 119,A -120.6275,B 24.9577,C -1.5025,E1 24.9274,E2 206.7442} C_DIS
LIN {X -54.9452,Y -103.4194,Z 119,A -121.8935,B 24.9577,C -1.5041,E1 24.9243,E2 208.0101} C_DIS
LIN {X -57.4667,Y -102.0398,Z 119,A -123.3039,B 24.9575,C -1.5058,E1 24.9208,E2 209.4204} C_DIS
LIN {X -59.9536,Y -100.5988,Z 119,A -124.7368,B 24.9575,C -1.5067,E1 24.9174,E2 210.8555} C_DIS
LIN {X -62.6539,Y -98.9413,Z 119,A -126.2698,B 24.9573,C -1.5098,E1 24.9137,E2 212.386} C_DIS
LIN {X -64.8988,Y -97.4822,Z 119,A -127.5949,B 24.9573,C -1.5113,E1 24.9107,E2 213.712} C_DIS
LIN {X -67.1917,Y -95.9158,Z 119,A -128.9342,B 24.957,C -1.5144,E1 24.9076,E2 215.0485} C_DIS
LIN {X -69.5253,Y -94.2379,Z 119,A -130.3591,B 24.957,C -1.516,E1 24.9044,E2 216.4745} C_DIS
LIN {X -71.7509,Y -92.5543,Z 119,A -131.7392,B 24.9568,C -1.5178,E1 24.9013,E2 217.8552} C_DIS
LIN {X -74.2942,Y -90.5277,Z 119,A -133.3272,B 24.9567,C -1.5209,E1 24.8979,E2 219.4419} C_DIS
LIN {X -76.2695,Y -88.868,Z 119,A -134.5676,B 24.9565,C -1.5243,E1 24.8952,E2 220.679} C_DIS
LIN {X -78.2976,Y -87.0857,Z 119,A -135.9726,B 24.9565,C -1.5234,E1 24.8923,E2 222.0918} C_DIS
LIN {X -80.7525,Y -84.817,Z 119,A -137.5643,B 24.9562,C -1.5286,E1 24.889,E2 223.6776} C_DIS
LIN {X -82.8097,Y -82.8097,Z 119,A -138.9769,B 24.9561,C -1.5313,E1 24.8862,E2 225.0897} C_DIS
LIN {X -84.6128,Y -80.9643,Z 119,A -140.2451,B 24.9559,C -1.5338,E1 24.8838,E2 226.3573} C_DIS
LIN {X -86.5743,Y -78.8634,Z 119,A -141.6581,B 24.9558,C -1.5367,E1 24.8811,E2 227.7698} C_DIS
LIN {X -88.6772,Y -76.4935,Z 119,A -143.216,B 24.9556,C -1.5399,E1 24.8782,E2 229.327} C_DIS
LIN {X -90.3397,Y -74.5204,Z 119,A -144.485,B 24.9554,C -1.5426,E1 24.876,E2 230.5954} C_DIS
LIN {X -92.3237,Y -72.0501,Z 119,A -146.0429,B 24.9552,C -1.546,E1 24.8733,E2 232.1525} C_DIS
LIN {X -94.0641,Y -69.7627,Z 119,A -147.4567,B 24.955,C -1.5492,E1 24.8709,E2 233.5656} C_DIS
LIN {X -95.4251,Y -67.8855,Z 119,A -148.6664,B 24.955,C -1.5489,E1 24.8689,E2 234.7819} C_DIS
LIN {X -97.2089,Y -65.3068,Z 119,A -150.1401,B 24.9547,C -1.5553,E1 24.8666,E2 236.2475} C_DIS
LIN {X -98.7824,Y -62.9015,Z 119,A -151.5542,B 24.9545,C -1.5587,E1 24.8645,E2 237.6608} C_DIS
LIN {X -100.235,Y -60.5592,Z 119,A -152.9512,B 24.9544,C -1.5603,E1 24.8624,E2 239.0612} C_DIS
LIN {X -101.8964,Y -57.7236,Z 119,A -154.5276,B 24.9541,C -1.5659,E1 24.8602,E2 240.6324} C_DIS
LIN {X -103.2823,Y -55.2055,Z 119,A -155.9422,B 24.9539,C -1.5694,E1 24.8583,E2 242.046} C_DIS
LIN {X -104.5304,Y -52.8023,Z 119,A -157.2678,B 24.9536,C -1.5731,E1 24.8567,E2 243.37} C_DIS
LIN {X -105.7393,Y -50.3364,Z 119,A -158.627,B 24.9534,C -1.5763,E1 24.855,E2 244.7289} C_DIS
LIN {X -106.9428,Y -47.7263,Z 119,A -160.012,B 24.9532,C -1.5812,E1 24.8534,E2 246.1098} C_DIS
LIN {X -108.0818,Y -45.0874,Z 119,A -161.4553,B 24.953,C -1.5838,E1 24.8518,E2 247.555} C_DIS
LIN {X -109.0682,Y -42.6443,Z 119,A -162.8189,B 24.953,C -1.5845,E1 24.8504,E2 248.9245} C_DIS
LIN {X -110.2648,Y -39.4534,Z 119,A -164.4324,B 24.9525,C -1.5916,E1 24.8489,E2 250.53} C_DIS
LIN {X -111.1998,Y -36.7355,Z 119,A -165.8478,B 24.9523,C -1.5955,E1 24.8476,E2 251.9444} C_DIS
LIN {X -111.9807,Y -34.2764,Z 119,A -167.1185,B 24.9521,C -1.599,E1 24.8466,E2 253.214} C_DIS
LIN {X -112.7882,Y -31.5179,Z 119,A -168.5339,B 24.9519,C -1.603,E1 24.8455,E2 254.6282} C_DIS
LIN {X -113.6009,Y -28.4555,Z 119,A -170.0945,B 24.9516,C -1.6073,E1 24.8444,E2 256.1875} C_DIS
LIN {X -114.2273,Y -25.8226,Z 119,A -171.4203,B 24.9513,C -1.6114,E1 24.8435,E2 257.5114} C_DIS
LIN {X -114.8603,Y -22.8471,Z 119,A -172.926,B 24.9511,C -1.6153,E1 24.8427,E2 259.0165} C_DIS
LIN {X -115.3049,Y -20.475,Z 119,A -174.1364,B 24.951,C -1.6179,E1 24.8421,E2 260.2281} C_DIS
LIN {X -115.843,Y -17.1837,Z 119,A -175.7578,B 24.9506,C -1.6235,E1 24.8414,E2 261.8458} C_DIS
LIN {X -116.1921,Y -14.6273,Z 119,A -177.0515,B 24.9504,C -1.6262,E1 24.8409,E2 263.1405} C_DIS
LIN {X -116.516,Y -11.7714,Z 119,A -178.445,B 24.9501,C -1.6313,E1 24.8405,E2 264.5304} C_DIS
LIN {X -116.7698,Y -8.9085,Z 119,A -179.8834,B 24.9499,C -1.6345,E1 24.8402,E2 265.9698} C_DIS
LIN {X -116.9533,Y -6.0401,Z 119,A 178.7038,B 24.9497,C -1.6388,E1 24.84,E2 267.3809} C_DIS
LIN {X -117.0753,Y -2.874,Z 119,A 177.0125,B 24.9497,C -1.638,E1 24.8398,E2 269.0841} C_DIS
LIN {X -117.1051,Y 0.9576,Z 119,A 175.2093,B 24.9492,C -1.6471,E1 24.8398,E2 270.8766} C_DIS
LIN {X -117.0403,Y 4.0165,Z 119,A 173.7664,B 24.9487,C -1.6541,E1 24.8399,E2 272.3114} C_DIS
LIN {X -116.8902,Y 7.1813,Z 119,A 172.2056,B 24.9484,C -1.6587,E1 24.8401,E2 273.8706} C_DIS
LIN {X -116.6787,Y 10.0478,Z 119,A 170.7893,B 24.9482,C -1.6629,E1 24.8405,E2 275.2855} C_DIS
LIN {X -116.397,Y 12.9082,Z 119,A 169.3733,B 24.9479,C -1.6671,E1 24.8409,E2 276.7} C_DIS
LIN {X -116.0452,Y 15.7608,Z 119,A 167.957,B 24.9477,C -1.6712,E1 24.8414,E2 278.1149} C_DIS
LIN {X -115.6684,Y 18.3132,Z 119,A 166.6634,B 24.9475,C -1.6741,E1 24.8419,E2 279.4094} C_DIS
LIN {X -115.1841,Y 21.1464,Z 119,A 165.2473,B 24.9472,C -1.6782,E1 24.8426,E2 280.8239} C_DIS
LIN {X -114.6305,Y 23.9667,Z 119,A 163.8312,B 24.947,C -1.6824,E1 24.8434,E2 282.2385} C_DIS
LIN {X -113.9416,Y 27.0593,Z 119,A 162.2925,B 24.9466,C -1.6878,E1 24.8444,E2 283.7734} C_DIS
LIN {X -113.3164,Y 29.5625,Z 119,A 160.9993,B 24.9464,C -1.6906,E1 24.8453,E2 285.0674} C_DIS
LIN {X -112.1515,Y 33.7134,Z 119,A 158.8975,B 24.946,C -1.6976,E1 24.8469,E2 287.1646} C_DIS
LIN {X -111.1998,Y 36.7354,Z 119,A 157.337,B 24.9457,C -1.7021,E1 24.8482,E2 288.7235} C_DIS
LIN {X -109.8731,Y 40.5271,Z 119,A 155.3358,B 24.9454,C -1.7068,E1 24.8501,E2 290.7248} C_DIS
LIN {X -108.8455,Y 43.2113,Z 119,A 153.9425,B 24.9451,C -1.7117,E1 24.8515,E2 292.1142} C_DIS
LIN {X -107.7522,Y 45.8695,Z 119,A 152.5268,B 24.9448,C -1.7156,E1 24.853,E2 293.5284} C_DIS
LIN {X -106.5941,Y 48.5001,Z 119,A 151.1298,B 24.9445,C -1.7203,E1 24.8546,E2 294.9219} C_DIS
LIN {X -105.3717,Y 51.1014,Z 119,A 149.6736,B 24.9444,C -1.7225,E1 24.8564,E2 296.3807} C_DIS
LIN {X -104.1116,Y 53.6216,Z 119,A 148.3025,B 24.9441,C -1.727,E1 24.8581,E2 297.7486} C_DIS
LIN {X -102.5971,Y 56.4688,Z 119,A 146.7207,B 24.9438,C -1.7314,E1 24.8602,E2 299.3282} C_DIS
LIN {X -101.1804,Y 58.9697,Z 119,A 145.3053,B 24.9436,C -1.7352,E1 24.8621,E2 300.7421} C_DIS
LIN {X -99.8555,Y 61.1836,Z 119,A 144.0351,B 24.9434,C -1.7385,E1 24.864,E2 302.0108} C_DIS
LIN {X -98.3733,Y 63.5387,Z 119,A 142.655,B 24.9432,C -1.7416,E1 24.866,E2 303.3904} C_DIS
LIN {X -96.8483,Y 65.8395,Z 119,A 141.2787,B 24.943,C -1.7444,E1 24.8682,E2 304.7671} C_DIS
LIN {X -95.084,Y 68.3636,Z 119,A 139.7685,B 24.9427,C -1.7484,E1 24.8706,E2 306.2751} C_DIS
LIN {X -93.3776,Y 70.6765,Z 119,A 138.3763,B 24.9424,C -1.7528,E1 24.8729,E2 307.6634} C_DIS
LIN {X -91.615,Y 72.9468,Z 119,A 136.9396,B 24.9423,C -1.7553,E1 24.8754,E2 309.101} C_DIS
LIN {X -89.6092,Y 75.3995,Z 119,A 135.4028,B 24.9419,C -1.7599,E1 24.8782,E2 310.6339} C_DIS
LIN {X -87.7318,Y 77.5759,Z 119,A 133.9887,B 24.9417,C -1.7632,E1 24.8808,E2 312.0465} C_DIS
LIN {X -85.8016,Y 79.7056,Z 119,A 132.575,B 24.9415,C -1.7665,E1 24.8834,E2 313.4587} C_DIS
LIN {X -84.0238,Y 81.5754,Z 119,A 131.3058,B 24.9413,C -1.7693,E1 24.8859,E2 314.7265} C_DIS
LIN {X -81.9966,Y 83.6129,Z 119,A 129.8922,B 24.9411,C -1.7725,E1 24.8887,E2 316.1387} C_DIS
LIN {X -79.9199,Y 85.6,Z 119,A 128.4787,B 24.9409,C -1.7755,E1 24.8915,E2 317.5508} C_DIS
LIN {X -77.7951,Y 87.5356,Z 119,A 127.0431,B 24.9408,C -1.7776,E1 24.8945,E2 318.9872} C_DIS
LIN {X -74.5204,Y 90.3397,Z 119,A 124.9235,B 24.9405,C -1.7819,E1 24.899,E2 321.1048} C_DIS
LIN {X -72.0501,Y 92.3237,Z 119,A 123.3883,B 24.9402,C -1.7858,E1 24.9024,E2 322.6361} C_DIS
LIN {X -69.7627,Y 94.0641,Z 119,A 121.9757,B 24.94,C -1.7885,E1 24.9055,E2 324.0474} C_DIS
LIN {X -67.4332,Y 95.7478,Z 119,A 120.5631,B 24.9399,C -1.7912,E1 24.9087,E2 325.4587} C_DIS
LIN {X -65.3068,Y 97.2089,Z 119,A 119.2953,B 24.9397,C -1.7935,E1 24.9117,E2 326.7253} C_DIS
LIN {X -62.9015,Y 98.7824,Z 119,A 117.8833,B 24.9395,C -1.7959,E1 24.915,E2 328.1359} C_DIS
LIN {X -60.4583,Y 100.2963,Z 119,A 116.4716,B 24.9394,C -1.7983,E1 24.9183,E2 329.5464} C_DIS
Enddeposition()
END
